LIN {X 0,Y 182.799,Z 411.389,A -85,B 0,C 180,E1 -25534.202,E2 -25534.202} C_VEL
LIN {X 0,Y 178.452,Z 402.819,A -85,B 0,C 180,E1 -25537.343,E2 -25537.343} C_VEL
LIN {X 0,Y 174.353,Z 395.574,A -85,B 0,C 180,E1 -25540.73,E2 -25540.73} C_VEL
LIN {X 0,Y 170.79,Z 389.828,A -85,B 0,C 180,E1 -25544.18,E2 -25544.18} C_VEL
LIN {X 0,Y 168.295,Z 385.886,A -85,B 0,C 180,E1 -25547.081,E2 -25547.081} C_VEL
LIN {X 0,Y 165.87,Z 382.031,A -85,B 0,C 180,E1 -25550.551,E2 -25550.551} C_VEL
LIN {X 0,Y 163.815,Z 378.873,A -85,B 0,C 180,E1 -25554.423,E2 -25554.423} C_VEL
LIN {X 0,Y 163.406,Z 377.726,A -85,B 0,C 180,E1 -25555.53,E2 -25555.53} C_VEL
LIN {X 0,Y 161.705,Z 376.148,A -85,B 0,C 180,E1 -25561.556,E2 -25561.556} C_VEL
LIN {X 0,Y 161.787,Z 376.62,A -85,B 0,C 180,E1 -25568.746,E2 -25568.746} C_VEL
LIN {X 0,Y 163.31,Z 378.032,A -85,B 0,C 180,E1 -25573.883,E2 -25573.883} C_VEL
LIN {X 0,Y 164.977,Z 381.356,A -85,B 0,C 180,E1 -25577.59,E2 -25577.59} C_VEL
LIN {X 0,Y 166.397,Z 382.961,A -85,B 0,C 180,E1 -25579.829,E2 -25579.829} C_VEL
LIN {X 0,Y 169.118,Z 387.647,A -85,B 0,C 180,E1 -25583.533,E2 -25583.533} C_VEL
LIN {X 0,Y 171.719,Z 392.777,A -85,B 0,C 180,E1 -25586.48,E2 -25586.48} C_VEL
LIN {X 0,Y 174.969,Z 399.659,A -85,B 0,C 180,E1 -25589.641,E2 -25589.641} C_VEL
LIN {X 0,Y 178.784,Z 408.58,A -85,B 0,C 180,E1 -25592.879,E2 -25592.879} C_VEL
LIN {X 0,Y 182.303,Z 418.101,A -85,B 0,C 180,E1 -25595.582,E2 -25595.582} C_VEL
LIN {X 0,Y 180.18,Z 440.666,A -85,B 0,C 180,E1 -25596.357,E2 -25596.357} C_VEL
LIN {X 0,Y 177.692,Z 453.902,A -85,B 0,C 180,E1 -25597.054,E2 -25597.054} C_VEL
LIN {X 0,Y 174.058,Z 466.777,A -85,B 0,C 180,E1 -25598.06,E2 -25598.06} C_VEL
LIN {X 0,Y 169.465,Z 479.095,A -85,B 0,C 180,E1 -25599.428,E2 -25599.428} C_VEL
LIN {X 0,Y 165.043,Z 488.832,A -85,B 0,C 180,E1 -25600.9,E2 -25600.9} C_VEL
LIN {X 0,Y 159.537,Z 499.053,A -85,B 0,C 180,E1 -25602.914,E2 -25602.914} C_VEL
LIN {X 0,Y 153.083,Z 509.068,A -85,B 0,C 180,E1 -25605.562,E2 -25605.562} C_VEL
LIN {X 0,Y 146.57,Z 517.891,A -85,B 0,C 180,E1 -25608.752,E2 -25608.752} C_VEL
LIN {X 0,Y 140.532,Z 524.996,A -85,B 0,C 180,E1 -25612.22,E2 -25612.22} C_VEL
LIN {X 0,Y 134.921,Z 530.971,A -85,B 0,C 180,E1 -25616.262,E2 -25616.262} C_VEL
LIN {X 0,Y 129.964,Z 535.823,A -85,B 0,C 180,E1 -25620.876,E2 -25620.876} C_VEL
LIN {X 0,Y 127.296,Z 538.125,A -85,B 0,C 180,E1 -25623.788,E2 -25623.788} C_VEL
LIN {X 0,Y 125.021,Z 540.003,A -85,B 0,C 180,E1 -25626.826,E2 -25626.826} C_VEL
LIN {X 0,Y 123.066,Z 541.427,A -85,B 0,C 180,E1 -25629.961,E2 -25629.961} C_VEL
LIN {X 0,Y 120.543,Z 543.117,A -85,B 0,C 180,E1 -25636.513,E2 -25636.513} C_VEL
LIN {X 0,Y 119.833,Z 543.394,A -85,B 0,C 180,E1 -25639.865,E2 -25639.865} C_VEL
LIN {X 0,Y 119.419,Z 543.249,A -85,B 0,C 180,E1 -25643.239,E2 -25643.239} C_VEL
LIN {X 0,Y 119.354,Z 542.709,A -85,B 0,C 180,E1 -25646.623,E2 -25646.623} C_VEL
LIN {X 0,Y 119.48,Z 541.653,A -85,B 0,C 180,E1 -25650.377,E2 -25650.377} C_VEL
LIN {X 0,Y 119.363,Z 540.421,A -85,B 0,C 180,E1 -25653.374,E2 -25653.374} C_VEL
LIN {X 0,Y 119.606,Z 537.522,A -85,B 0,C 180,E1 -25658.446,E2 -25658.446} C_VEL
LIN {X 0,Y 120.419,Z 533.561,A -85,B 0,C 180,E1 -25663.499,E2 -25663.499} C_VEL
LIN {X 0,Y 122.359,Z 527.446,A -85,B 0,C 180,E1 -25669.284,E2 -25669.284} C_VEL
LIN {X 0,Y 124.971,Z 520.737,A -85,B 0,C 180,E1 -25674.06,E2 -25674.06} C_VEL
LIN {X 0,Y 126.931,Z 516.144,A -85,B 0,C 180,E1 -25676.705,E2 -25676.705} C_VEL
LIN {X 0,Y 127.743,Z 512.422,A -85,B 0,C 180,E1 -25678.739,E2 -25678.739} C_VEL
LIN {X 0,Y 127.797,Z 505.991,A -85,B 0,C 180,E1 -25682.117,E2 -25682.117} C_VEL
LIN {X 0,Y 127.996,Z 499.009,A -85,B 0,C 180,E1 -25685.265,E2 -25685.265} C_VEL
LIN {X 0,Y 128.979,Z 494.425,A -85,B 0,C 180,E1 -25686.871,E2 -25686.871} C_VEL
LIN {X 0,Y 133.124,Z 482.951,A -85,B 0,C 180,E1 -25689.798,E2 -25689.798} C_VEL
LIN {X 0,Y 136.538,Z 471.516,A -85,B 0,C 180,E1 -25691.999,E2 -25691.999} C_VEL
LIN {X 0,Y 139.394,Z 459.785,A -85,B 0,C 180,E1 -25693.636,E2 -25693.636} C_VEL
LIN {X 0,Y 141.652,Z 446.808,A -85,B 0,C 180,E1 -25694.907,E2 -25694.907} C_VEL
LIN {X 0,Y 143.079,Z 433.332,A -85,B 0,C 180,E1 -25695.737,E2 -25695.737} C_VEL
LIN {X 0,Y 145.458,Z 398.287,A -85,B 0,C 180,E1 -25697.199,E2 -25697.199} C_VEL
LIN {X 0,Y 144.883,Z 389.327,A -85,B 0,C 180,E1 -25698.004,E2 -25698.004} C_VEL
LIN {X 0,Y 140.812,Z 377.368,A -85,B 0,C 180,E1 -25700.429,E2 -25700.429} C_VEL
LIN {X 0,Y 136.37,Z 367.095,A -85,B 0,C 180,E1 -25703.15,E2 -25703.15} C_VEL
LIN {X 0,Y 133.489,Z 362.113,A -85,B 0,C 180,E1 -25704.958,E2 -25704.958} C_VEL
LIN {X 0,Y 129.04,Z 355.347,A -85,B 0,C 180,E1 -25707.982,E2 -25707.982} C_VEL
LIN {X 0,Y 126.092,Z 351.147,A -85,B 0,C 180,E1 -25710.209,E2 -25710.209} C_VEL
LIN {X 0,Y 123.61,Z 347.782,A -85,B 0,C 180,E1 -25712.256,E2 -25712.256} C_VEL
LIN {X 0,Y 122.782,Z 346.727,A -85,B 0,C 180,E1 -25712.977,E2 -25712.977} C_VEL
LIN {X 0,Y 120.458,Z 344.175,A -85,B 0,C 180,E1 -25715.091,E2 -25715.091} C_VEL
LIN {X 0,Y 119.301,Z 341.838,A -85,B 0,C 180,E1 -25716.359,E2 -25716.359} C_VEL
LIN {X 0,Y 116.692,Z 339.986,A -85,B 0,C 180,E1 -25719.047,E2 -25719.047} C_VEL
LIN {X 0,Y 115.292,Z 337.525,A -85,B 0,C 180,E1 -25720.873,E2 -25720.873} C_VEL
LIN {X 0,Y 114.986,Z 336.158,A -85,B 0,C 180,E1 -25721.514,E2 -25721.514} C_VEL
LIN {X 0,Y 115.282,Z 336.094,A -85,B 0,C 180,E1 -25727.262,E2 -25727.262} C_VEL
LIN {X 0,Y 115.385,Z 336.109,A -85,B 0,C 180,E1 -25733.002,E2 -25733.002} C_VEL
LIN {X 0,Y 115.988,Z 336,A -85,B 0,C 180,E1 -25739.999,E2 -25739.999} C_VEL
LIN {X 0,Y 115.355,Z 336.095,A -85,B 0,C 180,E1 -25746.998,E2 -25746.998} C_VEL
LIN {X 0,Y 115.245,Z 336.108,A -85,B 0,C 180,E1 -25752.657,E2 -25752.657} C_VEL
LIN {X 0,Y 114.996,Z 336.138,A -85,B 0,C 180,E1 -25757.792,E2 -25757.792} C_VEL
LIN {X 0,Y 114.943,Z 336.152,A -85,B 0,C 180,E1 -25763.492,E2 -25763.492} C_VEL
LIN {X 0,Y 114.878,Z 336.207,A -85,B 0,C 180,E1 -25769.051,E2 -25769.051} C_VEL
LIN {X 0,Y 115.585,Z 338.454,A -85,B 0,C 180,E1 -25770.171,E2 -25770.171} C_VEL
LIN {X 0,Y 117.375,Z 340.759,A -85,B 0,C 180,E1 -25772.319,E2 -25772.319} C_VEL
LIN {X 0,Y 119.339,Z 342.102,A -85,B 0,C 180,E1 -25774.3,E2 -25774.3} C_VEL
LIN {X 0,Y 121.209,Z 345.34,A -85,B 0,C 180,E1 -25776.249,E2 -25776.249} C_VEL
LIN {X 0,Y 123.407,Z 347.522,A -85,B 0,C 180,E1 -25778.163,E2 -25778.163} C_VEL
LIN {X 0,Y 125.883,Z 351.047,A -85,B 0,C 180,E1 -25780.238,E2 -25780.238} C_VEL
LIN {X 0,Y 127.309,Z 353.048,A -85,B 0,C 180,E1 -25781.347,E2 -25781.347} C_VEL
LIN {X 0,Y 130.512,Z 357.56,A -85,B 0,C 180,E1 -25783.655,E2 -25783.655} C_VEL
LIN {X 0,Y 135.571,Z 365.369,A -85,B 0,C 180,E1 -25786.929,E2 -25786.929} C_VEL
LIN {X 0,Y 140.03,Z 373.18,A -85,B 0,C 180,E1 -25789.535,E2 -25789.535} C_VEL
LIN {X 0,Y 145.399,Z 384.296,A -85,B 0,C 180,E1 -25792.444,E2 -25792.444} C_VEL
LIN {X 0,Y 146.229,Z 386.228,A -85,B 0,C 180,E1 -25792.877,E2 -25792.877} C_VEL
LIN {X 0,Y 143.016,Z 431.95,A -85,B 0,C 180,E1 -25794.862,E2 -25794.862} C_VEL
LIN {X 0,Y 141.276,Z 445.448,A -85,B 0,C 180,E1 -25795.98,E2 -25795.98} C_VEL
LIN {X 0,Y 138.966,Z 457.681,A -85,B 0,C 180,E1 -25797.499,E2 -25797.499} C_VEL
LIN {X 0,Y 136.013,Z 468.763,A -85,B 0,C 180,E1 -25799.321,E2 -25799.321} C_VEL
LIN {X 0,Y 132.218,Z 480.314,A -85,B 0,C 180,E1 -25801.854,E2 -25801.854} C_VEL
LIN {X 0,Y 128.453,Z 490.68,A -85,B 0,C 180,E1 -25804.913,E2 -25804.913} C_VEL
LIN {X 0,Y 124.639,Z 500.01,A -85,B 0,C 180,E1 -25808.501,E2 -25808.501} C_VEL
LIN {X 0,Y 120.705,Z 509.025,A -85,B 0,C 180,E1 -25813.076,E2 -25813.076} C_VEL
LIN {X 0,Y 117.573,Z 516.285,A -85,B 0,C 180,E1 -25817.925,E2 -25817.925} C_VEL
LIN {X 0,Y 115.17,Z 522.106,A -85,B 0,C 180,E1 -25822.991,E2 -25822.991} C_VEL
LIN {X 0,Y 113.537,Z 526.693,A -85,B 0,C 180,E1 -25828.228,E2 -25828.228} C_VEL
LIN {X 0,Y 112.689,Z 530.291,A -85,B 0,C 180,E1 -25833.758,E2 -25833.758} C_VEL
LIN {X 0,Y 112.087,Z 533.325,A -85,B 0,C 180,E1 -25840.843,E2 -25840.843} C_VEL
LIN {X 0,Y 112.309,Z 534.286,A -85,B 0,C 180,E1 -25844.497,E2 -25844.497} C_VEL
LIN {X 0,Y 112.946,Z 534.841,A -85,B 0,C 180,E1 -25848.128,E2 -25848.128} C_VEL
LIN {X 0,Y 114.191,Z 534.925,A -85,B 0,C 180,E1 -25852.604,E2 -25852.604} C_VEL
LIN {X 0,Y 116.816,Z 534.015,A -85,B 0,C 180,E1 -25858.772,E2 -25858.772} C_VEL
LIN {X 0,Y 118.859,Z 532.918,A -85,B 0,C 180,E1 -25862.153,E2 -25862.153} C_VEL
LIN {X 0,Y 121.992,Z 530.899,A -85,B 0,C 180,E1 -25866.241,E2 -25866.241} C_VEL
LIN {X 0,Y 127.137,Z 526.951,A -85,B 0,C 180,E1 -25871.557,E2 -25871.557} C_VEL
LIN {X 0,Y 132.391,Z 522.293,A -85,B 0,C 180,E1 -25875.78,E2 -25875.78} C_VEL
LIN {X 0,Y 139.326,Z 515.206,A -85,B 0,C 180,E1 -25880.288,E2 -25880.288} C_VEL
LIN {X 0,Y 145.936,Z 507.482,A -85,B 0,C 180,E1 -25883.771,E2 -25883.771} C_VEL
LIN {X 0,Y 151.788,Z 499.51,A -85,B 0,C 180,E1 -25886.453,E2 -25886.453} C_VEL
LIN {X 0,Y 157.898,Z 489.721,A -85,B 0,C 180,E1 -25888.961,E2 -25888.961} C_VEL
LIN {X 0,Y 163.569,Z 478.78,A -85,B 0,C 180,E1 -25891.098,E2 -25891.098} C_VEL
LIN {X 0,Y 168.238,Z 467.913,A -85,B 0,C 180,E1 -25892.645,E2 -25892.645} C_VEL
LIN {X 0,Y 172.134,Z 456.207,A -85,B 0,C 180,E1 -25893.927,E2 -25893.927} C_VEL
LIN {X 0,Y 175.292,Z 443.368,A -85,B 0,C 180,E1 -25894.947,E2 -25894.947} C_VEL
LIN {X 0,Y 177.371,Z 430.99,A -85,B 0,C 180,E1 -25895.563,E2 -25895.563} C_VEL
LIN {X 0,Y 178.918,Z 414.661,A -85,B 0,C 180,E1 -25896.081,E2 -25896.081} C_VEL
LIN {X 0,Y 175.33,Z 407.397,A -85,B 0,C 180,E1 -25898.931,E2 -25898.931} C_VEL
LIN {X 0,Y 171.86,Z 400.977,A -85,B 0,C 180,E1 -25902.063,E2 -25902.063} C_VEL
LIN {X 0,Y 168.77,Z 395.843,A -85,B 0,C 180,E1 -25905.3,E2 -25905.3} C_VEL
LIN {X 0,Y 166.638,Z 392.303,A -85,B 0,C 180,E1 -25907.981,E2 -25907.981} C_VEL
LIN {X 0,Y 164.603,Z 388.858,A -85,B 0,C 180,E1 -25911.097,E2 -25911.097} C_VEL
LIN {X 0,Y 162.545,Z 385.367,A -85,B 0,C 180,E1 -25915.327,E2 -25915.327} C_VEL
LIN {X 0,Y 162.246,Z 384.661,A -85,B 0,C 180,E1 -25916.18,E2 -25916.18} C_VEL
LIN {X 0,Y 160.874,Z 383.217,A -85,B 0,C 180,E1 -25921.295,E2 -25921.295} C_VEL
LIN {X 0,Y 160.921,Z 383.691,A -85,B 0,C 180,E1 -25928.793,E2 -25928.793} C_VEL
LIN {X 0,Y 162.192,Z 384.921,A -85,B 0,C 180,E1 -25933.309,E2 -25933.309} C_VEL
LIN {X 0,Y 163.988,Z 388.453,A -85,B 0,C 180,E1 -25937.458,E2 -25937.458} C_VEL
LIN {X 0,Y 165.013,Z 389.709,A -85,B 0,C 180,E1 -25939.153,E2 -25939.153} C_VEL
LIN {X 0,Y 167.294,Z 393.779,A -85,B 0,C 180,E1 -25942.485,E2 -25942.485} C_VEL
LIN {X 0,Y 169.827,Z 399.15,A -85,B 0,C 180,E1 -25945.591,E2 -25945.591} C_VEL
LIN {X 0,Y 172.909,Z 406.19,A -85,B 0,C 180,E1 -25948.803,E2 -25948.803} C_VEL
LIN {X 0,Y 176.384,Z 414.842,A -85,B 0,C 180,E1 -25951.951,E2 -25951.951} C_VEL
LIN {X 0,Y 178.488,Z 420.805,A -85,B 0,C 180,E1 -25953.71,E2 -25953.71} C_VEL
LIN {X 0,Y 176.512,Z 440.736,A -85,B 0,C 180,E1 -25954.409,E2 -25954.409} C_VEL
LIN {X 0,Y 174.008,Z 453.597,A -85,B 0,C 180,E1 -25955.075,E2 -25955.075} C_VEL
LIN {X 0,Y 170.502,Z 465.847,A -85,B 0,C 180,E1 -25956.008,E2 -25956.008} C_VEL
LIN {X 0,Y 165.751,Z 478.298,A -85,B 0,C 180,E1 -25957.342,E2 -25957.342} C_VEL
LIN {X 0,Y 161.104,Z 488.137,A -85,B 0,C 180,E1 -25958.759,E2 -25958.759} C_VEL
LIN {X 0,Y 155.419,Z 498.431,A -85,B 0,C 180,E1 -25960.761,E2 -25960.761} C_VEL
LIN {X 0,Y 149.319,Z 507.707,A -85,B 0,C 180,E1 -25963.151,E2 -25963.151} C_VEL
LIN {X 0,Y 142.423,Z 516.71,A -85,B 0,C 180,E1 -25966.302,E2 -25966.302} C_VEL
LIN {X 0,Y 136.002,Z 523.988,A -85,B 0,C 180,E1 -25969.762,E2 -25969.762} C_VEL
LIN {X 0,Y 130.25,Z 529.843,A -85,B 0,C 180,E1 -25973.591,E2 -25973.591} C_VEL
LIN {X 0,Y 125.312,Z 534.478,A -85,B 0,C 180,E1 -25977.804,E2 -25977.804} C_VEL
LIN {X 0,Y 120.937,Z 538.031,A -85,B 0,C 180,E1 -25982.295,E2 -25982.295} C_VEL
LIN {X 0,Y 118.507,Z 539.861,A -85,B 0,C 180,E1 -25985.471,E2 -25985.471} C_VEL
LIN {X 0,Y 114.806,Z 542.26,A -85,B 0,C 180,E1 -25992.176,E2 -25992.176} C_VEL
LIN {X 0,Y 112.816,Z 543.129,A -85,B 0,C 180,E1 -25999.228,E2 -25999.228} C_VEL
LIN {X 0,Y 112.263,Z 542.379,A -85,B 0,C 180,E1 -26006.41,E2 -26006.41} C_VEL
LIN {X 0,Y 112.41,Z 541.423,A -85,B 0,C 180,E1 -26009.999,E2 -26009.999} C_VEL
LIN {X 0,Y 112.27,Z 540.031,A -85,B 0,C 180,E1 -26013.588,E2 -26013.588} C_VEL
LIN {X 0,Y 112.553,Z 537.082,A -85,B 0,C 180,E1 -26018.979,E2 -26018.979} C_VEL
LIN {X 0,Y 113.468,Z 533.061,A -85,B 0,C 180,E1 -26024.343,E2 -26024.343} C_VEL
LIN {X 0,Y 115.654,Z 526.854,A -85,B 0,C 180,E1 -26030.45,E2 -26030.45} C_VEL
LIN {X 0,Y 118.479,Z 520.07,A -85,B 0,C 180,E1 -26035.47,E2 -26035.47} C_VEL
LIN {X 0,Y 120.744,Z 514.832,A -85,B 0,C 180,E1 -26038.584,E2 -26038.584} C_VEL
LIN {X 0,Y 124.163,Z 506.59,A -85,B 0,C 180,E1 -26042.527,E2 -26042.527} C_VEL
LIN {X 0,Y 128.102,Z 496.752,A -85,B 0,C 180,E1 -26046.139,E2 -26046.139} C_VEL
LIN {X 0,Y 128.979,Z 494.425,A -85,B 0,C 180,E1 -26046.871,E2 -26046.871} C_VEL
LIN {X 0,Y 129.981,Z 489.751,A -85,B 0,C 180,E1 -26048.385,E2 -26048.385} C_VEL
LIN {X 0,Y 130.427,Z 478.545,A -85,B 0,C 180,E1 -26051.998,E2 -26051.998} C_VEL
LIN {X 0,Y 131.039,Z 471.722,A -85,B 0,C 180,E1 -26053.733,E2 -26053.733} C_VEL
LIN {X 0,Y 131.799,Z 468.136,A -85,B 0,C 180,E1 -26054.384,E2 -26054.384} C_VEL
LIN {X 0,Y 134.561,Z 456.507,A -85,B 0,C 180,E1 -26055.9,E2 -26055.9} C_VEL
LIN {X 0,Y 136.748,Z 443.617,A -85,B 0,C 180,E1 -26057.066,E2 -26057.066} C_VEL
LIN {X 0,Y 138.1,Z 429.088,A -85,B 0,C 180,E1 -26057.849,E2 -26057.849} C_VEL
LIN {X 0,Y 140.249,Z 399.102,A -85,B 0,C 180,E1 -26059.112,E2 -26059.112} C_VEL
LIN {X 0,Y 139.764,Z 391.546,A -85,B 0,C 180,E1 -26059.845,E2 -26059.845} C_VEL
LIN {X 0,Y 136.189,Z 380.798,A -85,B 0,C 180,E1 -26062.177,E2 -26062.177} C_VEL
LIN {X 0,Y 132.284,Z 371.453,A -85,B 0,C 180,E1 -26064.803,E2 -26064.803} C_VEL
LIN {X 0,Y 128.572,Z 364.909,A -85,B 0,C 180,E1 -26067.388,E2 -26067.388} C_VEL
LIN {X 0,Y 123.204,Z 356.965,A -85,B 0,C 180,E1 -26071.578,E2 -26071.578} C_VEL
LIN {X 0,Y 120.254,Z 352.917,A -85,B 0,C 180,E1 -26074.235,E2 -26074.235} C_VEL
LIN {X 0,Y 117.75,Z 349.777,A -85,B 0,C 180,E1 -26076.744,E2 -26076.744} C_VEL
LIN {X 0,Y 116.931,Z 348.248,A -85,B 0,C 180,E1 -26077.702,E2 -26077.702} C_VEL
LIN {X 0,Y 114.396,Z 345.983,A -85,B 0,C 180,E1 -26080.601,E2 -26080.601} C_VEL
LIN {X 0,Y 112.753,Z 342.88,A -85,B 0,C 180,E1 -26083.011,E2 -26083.011} C_VEL
LIN {X 0,Y 110.318,Z 341.255,A -85,B 0,C 180,E1 -26086.679,E2 -26086.679} C_VEL
LIN {X 0,Y 108.645,Z 338.426,A -85,B 0,C 180,E1 -26090.223,E2 -26090.223} C_VEL
LIN {X 0,Y 108.294,Z 336.972,A -85,B 0,C 180,E1 -26091.485,E2 -26091.485} C_VEL
LIN {X 0,Y 108.914,Z 336.88,A -85,B 0,C 180,E1 -26099.999,E2 -26099.999} C_VEL
LIN {X 0,Y 108.295,Z 336.968,A -85,B 0,C 180,E1 -26107.457,E2 -26107.457} C_VEL
LIN {X 0,Y 108.166,Z 336.991,A -85,B 0,C 180,E1 -26112.947,E2 -26112.947} C_VEL
LIN {X 0,Y 107.935,Z 337.086,A -85,B 0,C 180,E1 -26118.507,E2 -26118.507} C_VEL
LIN {X 0,Y 108.493,Z 339.139,A -85,B 0,C 180,E1 -26120.252,E2 -26120.252} C_VEL
LIN {X 0,Y 110.772,Z 341.962,A -85,B 0,C 180,E1 -26124.743,E2 -26124.743} C_VEL
LIN {X 0,Y 112.832,Z 343.115,A -85,B 0,C 180,E1 -26127.723,E2 -26127.723} C_VEL
LIN {X 0,Y 114.487,Z 346.252,A -85,B 0,C 180,E1 -26130.13,E2 -26130.13} C_VEL
LIN {X 0,Y 117.162,Z 348.772,A -85,B 0,C 180,E1 -26133.176,E2 -26133.176} C_VEL
LIN {X 0,Y 119.418,Z 352.183,A -85,B 0,C 180,E1 -26135.589,E2 -26135.589} C_VEL
LIN {X 0,Y 120.903,Z 353.816,A -85,B 0,C 180,E1 -26136.971,E2 -26136.971} C_VEL
LIN {X 0,Y 124.336,Z 358.803,A -85,B 0,C 180,E1 -26139.982,E2 -26139.982} C_VEL
LIN {X 0,Y 127.719,Z 363.738,A -85,B 0,C 180,E1 -26142.597,E2 -26142.597} C_VEL
LIN {X 0,Y 132.879,Z 372.086,A -85,B 0,C 180,E1 -26146.145,E2 -26146.145} C_VEL
LIN {X 0,Y 137.922,Z 381.827,A -85,B 0,C 180,E1 -26149.265,E2 -26149.265} C_VEL
LIN {X 0,Y 140.92,Z 388.415,A -85,B 0,C 180,E1 -26150.994,E2 -26150.994} C_VEL
LIN {X 0,Y 137.765,Z 431.864,A -85,B 0,C 180,E1 -26152.923,E2 -26152.923} C_VEL
LIN {X 0,Y 135.883,Z 445.712,A -85,B 0,C 180,E1 -26154.08,E2 -26154.08} C_VEL
LIN {X 0,Y 133.291,Z 458.5,A -85,B 0,C 180,E1 -26155.702,E2 -26155.702} C_VEL
LIN {X 0,Y 129.968,Z 470.244,A -85,B 0,C 180,E1 -26157.726,E2 -26157.726} C_VEL
LIN {X 0,Y 126.005,Z 481.573,A -85,B 0,C 180,E1 -26160.331,E2 -26160.331} C_VEL
LIN {X 0,Y 122.09,Z 491.743,A -85,B 0,C 180,E1 -26163.507,E2 -26163.507} C_VEL
LIN {X 0,Y 118.063,Z 500.901,A -85,B 0,C 180,E1 -26167.238,E2 -26167.238} C_VEL
LIN {X 0,Y 113.94,Z 509.809,A -85,B 0,C 180,E1 -26172.038,E2 -26172.038} C_VEL
LIN {X 0,Y 110.662,Z 516.974,A -85,B 0,C 180,E1 -26177.158,E2 -26177.158} C_VEL
LIN {X 0,Y 108.104,Z 522.698,A -85,B 0,C 180,E1 -26182.53,E2 -26182.53} C_VEL
LIN {X 0,Y 106.447,Z 527.205,A -85,B 0,C 180,E1 -26188.11,E2 -26188.11} C_VEL
LIN {X 0,Y 105.567,Z 530.644,A -85,B 0,C 180,E1 -26193.819,E2 -26193.819} C_VEL
LIN {X 0,Y 105.055,Z 532.379,A -85,B 0,C 180,E1 -26197.69,E2 -26197.69} C_VEL
LIN {X 0,Y 104.998,Z 533.704,A -85,B 0,C 180,E1 -26201.585,E2 -26201.585} C_VEL
LIN {X 0,Y 105.322,Z 534.634,A -85,B 0,C 180,E1 -26205.482,E2 -26205.482} C_VEL
LIN {X 0,Y 106.071,Z 535.129,A -85,B 0,C 180,E1 -26209.348,E2 -26209.348} C_VEL
LIN {X 0,Y 107.289,Z 535.201,A -85,B 0,C 180,E1 -26213.5,E2 -26213.5} C_VEL
LIN {X 0,Y 110.485,Z 534.205,A -85,B 0,C 180,E1 -26220.591,E2 -26220.591} C_VEL
LIN {X 0,Y 112.759,Z 533.046,A -85,B 0,C 180,E1 -26224.123,E2 -26224.123} C_VEL
LIN {X 0,Y 115.751,Z 531.262,A -85,B 0,C 180,E1 -26227.879,E2 -26227.879} C_VEL
LIN {X 0,Y 120.049,Z 528.247,A -85,B 0,C 180,E1 -26232.319,E2 -26232.319} C_VEL
LIN {X 0,Y 125.453,Z 523.919,A -85,B 0,C 180,E1 -26236.743,E2 -26236.743} C_VEL
LIN {X 0,Y 131.545,Z 518.352,A -85,B 0,C 180,E1 -26240.778,E2 -26240.778} C_VEL
LIN {X 0,Y 138.205,Z 511.354,A -85,B 0,C 180,E1 -26244.453,E2 -26244.453} C_VEL
LIN {X 0,Y 145.264,Z 502.723,A -85,B 0,C 180,E1 -26247.689,E2 -26247.689} C_VEL
LIN {X 0,Y 151.723,Z 493.408,A -85,B 0,C 180,E1 -26250.289,E2 -26250.289} C_VEL
LIN {X 0,Y 157.531,Z 483.314,A -85,B 0,C 180,E1 -26252.461,E2 -26252.461} C_VEL
LIN {X 0,Y 162.918,Z 472.021,A -85,B 0,C 180,E1 -26254.226,E2 -26254.226} C_VEL
LIN {X 0,Y 167.338,Z 460.287,A -85,B 0,C 180,E1 -26255.622,E2 -26255.622} C_VEL
LIN {X 0,Y 170.766,Z 448.312,A -85,B 0,C 180,E1 -26256.672,E2 -26256.672} C_VEL
LIN {X 0,Y 173.271,Z 435.759,A -85,B 0,C 180,E1 -26257.414,E2 -26257.414} C_VEL
LIN {X 0,Y 175.332,Z 418.304,A -85,B 0,C 180,E1 -26257.949,E2 -26257.949} C_VEL
LIN {X 0,Y 172.367,Z 411.99,A -85,B 0,C 180,E1 -26260.557,E2 -26260.557} C_VEL
LIN {X 0,Y 168.917,Z 405.563,A -85,B 0,C 180,E1 -26264,E2 -26264} C_VEL
LIN {X 0,Y 166.702,Z 401.685,A -85,B 0,C 180,E1 -26266.593,E2 -26266.593} C_VEL
LIN {X 0,Y 164.993,Z 398.634,A -85,B 0,C 180,E1 -26268.95,E2 -26268.95} C_VEL
LIN {X 0,Y 163.144,Z 395.409,A -85,B 0,C 180,E1 -26272.017,E2 -26272.017} C_VEL
LIN {X 0,Y 161.098,Z 391.549,A -85,B 0,C 180,E1 -26276.875,E2 -26276.875} C_VEL
LIN {X 0,Y 159.836,Z 390.177,A -85,B 0,C 180,E1 -26282.521,E2 -26282.521} C_VEL
LIN {X 0,Y 160.055,Z 390.765,A -85,B 0,C 180,E1 -26288.841,E2 -26288.841} C_VEL
LIN {X 0,Y 161.104,Z 391.812,A -85,B 0,C 180,E1 -26292.759,E2 -26292.759} C_VEL
LIN {X 0,Y 162.762,Z 395.265,A -85,B 0,C 180,E1 -26296.888,E2 -26296.888} C_VEL
LIN {X 0,Y 163.785,Z 396.679,A -85,B 0,C 180,E1 -26298.693,E2 -26298.693} C_VEL
LIN {X 0,Y 165.626,Z 400.165,A -85,B 0,C 180,E1 -26301.562,E2 -26301.562} C_VEL
LIN {X 0,Y 167.894,Z 405.33,A -85,B 0,C 180,E1 -26304.582,E2 -26304.582} C_VEL
LIN {X 0,Y 170.782,Z 412.392,A -85,B 0,C 180,E1 -26307.828,E2 -26307.828} C_VEL
LIN {X 0,Y 173.668,Z 420.159,A -85,B 0,C 180,E1 -26310.669,E2 -26310.669} C_VEL
LIN {X 0,Y 174.857,Z 423.716,A -85,B 0,C 180,E1 -26311.765,E2 -26311.765} C_VEL
LIN {X 0,Y 173.004,Z 441.112,A -85,B 0,C 180,E1 -26312.39,E2 -26312.39} C_VEL
LIN {X 0,Y 170.551,Z 453.173,A -85,B 0,C 180,E1 -26312.996,E2 -26312.996} C_VEL
LIN {X 0,Y 167.166,Z 464.912,A -85,B 0,C 180,E1 -26313.866,E2 -26313.866} C_VEL
LIN {X 0,Y 162.263,Z 477.507,A -85,B 0,C 180,E1 -26315.162,E2 -26315.162} C_VEL
LIN {X 0,Y 156.785,Z 488.729,A -85,B 0,C 180,E1 -26316.749,E2 -26316.749} C_VEL
LIN {X 0,Y 150.895,Z 498.851,A -85,B 0,C 180,E1 -26318.726,E2 -26318.726} C_VEL
LIN {X 0,Y 144.577,Z 507.983,A -85,B 0,C 180,E1 -26321.107,E2 -26321.107} C_VEL
LIN {X 0,Y 137.386,Z 516.896,A -85,B 0,C 180,E1 -26324.26,E2 -26324.26} C_VEL
LIN {X 0,Y 130.651,Z 524.094,A -85,B 0,C 180,E1 -26327.746,E2 -26327.746} C_VEL
LIN {X 0,Y 124.605,Z 529.866,A -85,B 0,C 180,E1 -26331.652,E2 -26331.652} C_VEL
LIN {X 0,Y 119.338,Z 534.437,A -85,B 0,C 180,E1 -26335.98,E2 -26335.98} C_VEL
LIN {X 0,Y 114.675,Z 537.937,A -85,B 0,C 180,E1 -26340.639,E2 -26340.639} C_VEL
LIN {X 0,Y 112.071,Z 539.713,A -85,B 0,C 180,E1 -26343.96,E2 -26343.96} C_VEL
LIN {X 0,Y 108.026,Z 542.059,A -85,B 0,C 180,E1 -26351.016,E2 -26351.016} C_VEL
LIN {X 0,Y 106.74,Z 542.663,A -85,B 0,C 180,E1 -26354.729,E2 -26354.729} C_VEL
LIN {X 0,Y 105.83,Z 542.852,A -85,B 0,C 180,E1 -26358.507,E2 -26358.507} C_VEL
LIN {X 0,Y 105.181,Z 542.05,A -85,B 0,C 180,E1 -26366.167,E2 -26366.167} C_VEL
LIN {X 0,Y 105.335,Z 541.069,A -85,B 0,C 180,E1 -26369.999,E2 -26369.999} C_VEL
LIN {X 0,Y 105.189,Z 539.627,A -85,B 0,C 180,E1 -26373.83,E2 -26373.83} C_VEL
LIN {X 0,Y 105.526,Z 536.63,A -85,B 0,C 180,E1 -26379.583,E2 -26379.583} C_VEL
LIN {X 0,Y 106.553,Z 532.548,A -85,B 0,C 180,E1 -26385.296,E2 -26385.296} C_VEL
LIN {X 0,Y 109.011,Z 526.263,A -85,B 0,C 180,E1 -26391.758,E2 -26391.758} C_VEL
LIN {X 0,Y 112.082,Z 519.405,A -85,B 0,C 180,E1 -26397.038,E2 -26397.038} C_VEL
LIN {X 0,Y 113.965,Z 515.38,A -85,B 0,C 180,E1 -26399.559,E2 -26399.559} C_VEL
LIN {X 0,Y 116.695,Z 509.196,A -85,B 0,C 180,E1 -26402.82,E2 -26402.82} C_VEL
LIN {X 0,Y 120.683,Z 500.042,A -85,B 0,C 180,E1 -26406.647,E2 -26406.647} C_VEL
LIN {X 0,Y 124.706,Z 489.923,A -85,B 0,C 180,E1 -26409.869,E2 -26409.869} C_VEL
LIN {X 0,Y 128.699,Z 478.671,A -85,B 0,C 180,E1 -26412.512,E2 -26412.512} C_VEL
LIN {X 0,Y 131.799,Z 468.136,A -85,B 0,C 180,E1 -26414.384,E2 -26414.384} C_VEL
LIN {X 0,Y 132.665,Z 462.724,A -85,B 0,C 180,E1 -26415.344,E2 -26415.344} C_VEL
LIN {X 0,Y 132.409,Z 453.764,A -85,B 0,C 180,E1 -26417.214,E2 -26417.214} C_VEL
LIN {X 0,Y 131.857,Z 444.61,A -85,B 0,C 180,E1 -26418.866,E2 -26418.866} C_VEL
LIN {X 0,Y 132.148,Z 438.863,A -85,B 0,C 180,E1 -26419.443,E2 -26419.443} C_VEL
LIN {X 0,Y 135.166,Z 400.629,A -85,B 0,C 180,E1 -26421.128,E2 -26421.128} C_VEL
LIN {X 0,Y 134.874,Z 393.98,A -85,B 0,C 180,E1 -26421.764,E2 -26421.764} C_VEL
LIN {X 0,Y 131.49,Z 383.608,A -85,B 0,C 180,E1 -26424.203,E2 -26424.203} C_VEL
LIN {X 0,Y 127.847,Z 374.792,A -85,B 0,C 180,E1 -26426.916,E2 -26426.916} C_VEL
LIN {X 0,Y 123.215,Z 366.999,A -85,B 0,C 180,E1 -26430.538,E2 -26430.538} C_VEL
LIN {X 0,Y 120.137,Z 362.449,A -85,B 0,C 180,E1 -26433.244,E2 -26433.244} C_VEL
LIN {X 0,Y 117.838,Z 359.099,A -85,B 0,C 180,E1 -26435.505,E2 -26435.505} C_VEL
LIN {X 0,Y 115.279,Z 355.624,A -85,B 0,C 180,E1 -26438.308,E2 -26438.308} C_VEL
LIN {X 0,Y 114.397,Z 354.432,A -85,B 0,C 180,E1 -26439.371,E2 -26439.371} C_VEL
LIN {X 0,Y 111.953,Z 351.561,A -85,B 0,C 180,E1 -26442.562,E2 -26442.562} C_VEL
LIN {X 0,Y 110.826,Z 349.535,A -85,B 0,C 180,E1 -26444.364,E2 -26444.364} C_VEL
LIN {X 0,Y 108.505,Z 347.495,A -85,B 0,C 180,E1 -26448.321,E2 -26448.321} C_VEL
LIN {X 0,Y 107.036,Z 344.518,A -85,B 0,C 180,E1 -26451.979,E2 -26451.979} C_VEL
LIN {X 0,Y 106.705,Z 343.89,A -85,B 0,C 180,E1 -26452.953,E2 -26452.953} C_VEL
LIN {X 0,Y 104.856,Z 342.696,A -85,B 0,C 180,E1 -26459.999,E2 -26459.999} C_VEL
LIN {X 0,Y 105.075,Z 343.36,A -85,B 0,C 180,E1 -26472.158,E2 -26472.158} C_VEL
LIN {X 0,Y 106.571,Z 344.146,A -85,B 0,C 180,E1 -26477.386,E2 -26477.386} C_VEL
LIN {X 0,Y 107.564,Z 346.607,A -85,B 0,C 180,E1 -26480.31,E2 -26480.31} C_VEL
LIN {X 0,Y 109.848,Z 349.097,A -85,B 0,C 180,E1 -26484.764,E2 -26484.764} C_VEL
LIN {X 0,Y 111.023,Z 349.852,A -85,B 0,C 180,E1 -26486.555,E2 -26486.555} C_VEL
LIN {X 0,Y 112.975,Z 353.182,A -85,B 0,C 180,E1 -26489.499,E2 -26489.499} C_VEL
LIN {X 0,Y 115.007,Z 355.245,A -85,B 0,C 180,E1 -26491.958,E2 -26491.958} C_VEL
LIN {X 0,Y 117.655,Z 359.003,A -85,B 0,C 180,E1 -26494.916,E2 -26494.916} C_VEL
LIN {X 0,Y 121.315,Z 364.264,A -85,B 0,C 180,E1 -26498.431,E2 -26498.431} C_VEL
LIN {X 0,Y 125.767,Z 371.178,A -85,B 0,C 180,E1 -26502.11,E2 -26502.11} C_VEL
LIN {X 0,Y 130.763,Z 380.001,A -85,B 0,C 180,E1 -26505.719,E2 -26505.719} C_VEL
LIN {X 0,Y 135.623,Z 390.455,A -85,B 0,C 180,E1 -26508.898,E2 -26508.898} C_VEL
LIN {X 0,Y 135.813,Z 391.21,A -85,B 0,C 180,E1 -26509.04,E2 -26509.04} C_VEL
LIN {X 0,Y 132.666,Z 431.76,A -85,B 0,C 180,E1 -26510.833,E2 -26510.833} C_VEL
LIN {X 0,Y 130.812,Z 445.029,A -85,B 0,C 180,E1 -26511.935,E2 -26511.935} C_VEL
LIN {X 0,Y 128.349,Z 457.153,A -85,B 0,C 180,E1 -26513.455,E2 -26513.455} C_VEL
LIN {X 0,Y 125.109,Z 468.525,A -85,B 0,C 180,E1 -26515.337,E2 -26515.337} C_VEL
LIN {X 0,Y 120.887,Z 480.231,A -85,B 0,C 180,E1 -26517.963,E2 -26517.963} C_VEL
LIN {X 0,Y 116.682,Z 490.7,A -85,B 0,C 180,E1 -26521.195,E2 -26521.195} C_VEL
LIN {X 0,Y 112.387,Z 500.146,A -85,B 0,C 180,E1 -26525.034,E2 -26525.034} C_VEL
LIN {X 0,Y 107.899,Z 509.233,A -85,B 0,C 180,E1 -26530.005,E2 -26530.005} C_VEL
LIN {X 0,Y 104.283,Z 516.55,A -85,B 0,C 180,E1 -26535.363,E2 -26535.363} C_VEL
LIN {X 0,Y 101.048,Z 523.272,A -85,B 0,C 180,E1 -26542.006,E2 -26542.006} C_VEL
LIN {X 0,Y 99.356,Z 527.706,A -85,B 0,C 180,E1 -26547.975,E2 -26547.975} C_VEL
LIN {X 0,Y 98.395,Z 531.084,A -85,B 0,C 180,E1 -26554.097,E2 -26554.097} C_VEL
LIN {X 0,Y 97.921,Z 532.787,A -85,B 0,C 180,E1 -26558.254,E2 -26558.254} C_VEL
LIN {X 0,Y 97.938,Z 534.081,A -85,B 0,C 180,E1 -26562.433,E2 -26562.433} C_VEL
LIN {X 0,Y 98.375,Z 534.97,A -85,B 0,C 180,E1 -26566.606,E2 -26566.606} C_VEL
LIN {X 0,Y 100.457,Z 535.474,A -85,B 0,C 180,E1 -26574.567,E2 -26574.567} C_VEL
LIN {X 0,Y 102.168,Z 535.132,A -85,B 0,C 180,E1 -26578.786,E2 -26578.786} C_VEL
LIN {X 0,Y 104.264,Z 534.381,A -85,B 0,C 180,E1 -26582.634,E2 -26582.634} C_VEL
LIN {X 0,Y 109.592,Z 531.637,A -85,B 0,C 180,E1 -26589.688,E2 -26589.688} C_VEL
LIN {X 0,Y 114.763,Z 528.279,A -85,B 0,C 180,E1 -26594.77,E2 -26594.77} C_VEL
LIN {X 0,Y 120.58,Z 523.88,A -85,B 0,C 180,E1 -26599.264,E2 -26599.264} C_VEL
LIN {X 0,Y 127.046,Z 518.235,A -85,B 0,C 180,E1 -26603.334,E2 -26603.334} C_VEL
LIN {X 0,Y 134.1,Z 511.116,A -85,B 0,C 180,E1 -26606.987,E2 -26606.987} C_VEL
LIN {X 0,Y 141.71,Z 502.1,A -85,B 0,C 180,E1 -26610.269,E2 -26610.269} C_VEL
LIN {X 0,Y 148.252,Z 492.93,A -85,B 0,C 180,E1 -26612.731,E2 -26612.731} C_VEL
LIN {X 0,Y 154.284,Z 482.601,A -85,B 0,C 180,E1 -26614.872,E2 -26614.872} C_VEL
LIN {X 0,Y 159.764,Z 471.385,A -85,B 0,C 180,E1 -26616.528,E2 -26616.528} C_VEL
LIN {X 0,Y 164.107,Z 460.043,A -85,B 0,C 180,E1 -26617.834,E2 -26617.834} C_VEL
LIN {X 0,Y 167.787,Z 447.319,A -85,B 0,C 180,E1 -26618.884,E2 -26618.884} C_VEL
LIN {X 0,Y 170.335,Z 434.321,A -85,B 0,C 180,E1 -26619.593,E2 -26619.593} C_VEL
LIN {X 0,Y 171.87,Z 421.656,A -85,B 0,C 180,E1 -26619.97,E2 -26619.97} C_VEL
LIN {X 0,Y 168.557,Z 414.703,A -85,B 0,C 180,E1 -26623.265,E2 -26623.265} C_VEL
LIN {X 0,Y 165.476,Z 408.852,A -85,B 0,C 180,E1 -26626.9,E2 -26626.9} C_VEL
LIN {X 0,Y 163.485,Z 405.173,A -85,B 0,C 180,E1 -26629.786,E2 -26629.786} C_VEL
LIN {X 0,Y 161.959,Z 402.243,A -85,B 0,C 180,E1 -26632.52,E2 -26632.52} C_VEL
LIN {X 0,Y 160.113,Z 398.537,A -85,B 0,C 180,E1 -26637.17,E2 -26637.17} C_VEL
LIN {X 0,Y 158.963,Z 397.225,A -85,B 0,C 180,E1 -26642.535,E2 -26642.535} C_VEL
LIN {X 0,Y 159.189,Z 397.837,A -85,B 0,C 180,E1 -26648.89,E2 -26648.89} C_VEL
LIN {X 0,Y 160.098,Z 398.901,A -85,B 0,C 180,E1 -26652.446,E2 -26652.446} C_VEL
LIN {X 0,Y 161.709,Z 402.244,A -85,B 0,C 180,E1 -26656.607,E2 -26656.607} C_VEL
LIN {X 0,Y 162.451,Z 403.433,A -85,B 0,C 180,E1 -26658.013,E2 -26658.013} C_VEL
LIN {X 0,Y 163.955,Z 406.431,A -85,B 0,C 180,E1 -26660.547,E2 -26660.547} C_VEL
LIN {X 0,Y 166.071,Z 411.647,A -85,B 0,C 180,E1 -26663.623,E2 -26663.623} C_VEL
LIN {X 0,Y 168.97,Z 419.289,A -85,B 0,C 180,E1 -26667.123,E2 -26667.123} C_VEL
LIN {X 0,Y 171.43,Z 426.611,A -85,B 0,C 180,E1 -26669.736,E2 -26669.736} C_VEL
LIN {X 0,Y 169.67,Z 441.805,A -85,B 0,C 180,E1 -26670.303,E2 -26670.303} C_VEL
LIN {X 0,Y 167,Z 454.164,A -85,B 0,C 180,E1 -26670.936,E2 -26670.936} C_VEL
LIN {X 0,Y 163.341,Z 465.974,A -85,B 0,C 180,E1 -26671.812,E2 -26671.812} C_VEL
LIN {X 0,Y 158.303,Z 478.292,A -85,B 0,C 180,E1 -26673.073,E2 -26673.073} C_VEL
LIN {X 0,Y 152.671,Z 489.312,A -85,B 0,C 180,E1 -26674.628,E2 -26674.628} C_VEL
LIN {X 0,Y 146.574,Z 499.236,A -85,B 0,C 180,E1 -26676.569,E2 -26676.569} C_VEL
LIN {X 0,Y 140.013,Z 508.26,A -85,B 0,C 180,E1 -26678.919,E2 -26678.919} C_VEL
LIN {X 0,Y 132.543,Z 517.082,A -85,B 0,C 180,E1 -26682.068,E2 -26682.068} C_VEL
LIN {X 0,Y 125.491,Z 524.186,A -85,B 0,C 180,E1 -26685.568,E2 -26685.568} C_VEL
LIN {X 0,Y 119.108,Z 529.875,A -85,B 0,C 180,E1 -26689.528,E2 -26689.528} C_VEL
LIN {X 0,Y 114.101,Z 533.902,A -85,B 0,C 180,E1 -26693.399,E2 -26693.399} C_VEL
LIN {X 0,Y 108.527,Z 537.834,A -85,B 0,C 180,E1 -26698.796,E2 -26698.796} C_VEL
LIN {X 0,Y 103.262,Z 540.905,A -85,B 0,C 180,E1 -26705.897,E2 -26705.897} C_VEL
LIN {X 0,Y 99.864,Z 542.427,A -85,B 0,C 180,E1 -26713.649,E2 -26713.649} C_VEL
LIN {X 0,Y 98.873,Z 542.574,A -85,B 0,C 180,E1 -26717.686,E2 -26717.686} C_VEL
LIN {X 0,Y 98.091,Z 541.721,A -85,B 0,C 180,E1 -26725.89,E2 -26725.89} C_VEL
LIN {X 0,Y 98.246,Z 540.713,A -85,B 0,C 180,E1 -26729.999,E2 -26729.999} C_VEL
LIN {X 0,Y 98.1,Z 539.218,A -85,B 0,C 180,E1 -26734.107,E2 -26734.107} C_VEL
LIN {X 0,Y 98.502,Z 536.164,A -85,B 0,C 180,E1 -26740.273,E2 -26740.273} C_VEL
LIN {X 0,Y 99.685,Z 532.021,A -85,B 0,C 180,E1 -26746.378,E2 -26746.378} C_VEL
LIN {X 0,Y 102.417,Z 525.67,A -85,B 0,C 180,E1 -26753.238,E2 -26753.238} C_VEL
LIN {X 0,Y 105.789,Z 518.741,A -85,B 0,C 180,E1 -26758.791,E2 -26758.791} C_VEL
LIN {X 0,Y 109.095,Z 511.739,A -85,B 0,C 180,E1 -26763.124,E2 -26763.124} C_VEL
LIN {X 0,Y 113.213,Z 503.076,A -85,B 0,C 180,E1 -26767.246,E2 -26767.246} C_VEL
LIN {X 0,Y 117.78,Z 492.468,A -85,B 0,C 180,E1 -26771.022,E2 -26771.022} C_VEL
LIN {X 0,Y 121.917,Z 481.984,A -85,B 0,C 180,E1 -26773.766,E2 -26773.766} C_VEL
LIN {X 0,Y 125.705,Z 470.436,A -85,B 0,C 180,E1 -26776.038,E2 -26776.038} C_VEL
LIN {X 0,Y 128.848,Z 458.466,A -85,B 0,C 180,E1 -26777.709,E2 -26777.709} C_VEL
LIN {X 0,Y 131.4,Z 444.815,A -85,B 0,C 180,E1 -26779.027,E2 -26779.027} C_VEL
LIN {X 0,Y 132.148,Z 438.863,A -85,B 0,C 180,E1 -26779.443,E2 -26779.443} C_VEL
LIN {X 0,Y 132.384,Z 433.087,A -85,B 0,C 180,E1 -26779.947,E2 -26779.947} C_VEL
LIN {X 0,Y 129.86,Z 414.309,A -85,B 0,C 180,E1 -26782.533,E2 -26782.533} C_VEL
LIN {X 0,Y 129.782,Z 408.483,A -85,B 0,C 180,E1 -26783.015,E2 -26783.015} C_VEL
LIN {X 0,Y 130.311,Z 399.937,A -85,B 0,C 180,E1 -26783.452,E2 -26783.452} C_VEL
LIN {X 0,Y 130.047,Z 396.241,A -85,B 0,C 180,E1 -26783.888,E2 -26783.888} C_VEL
LIN {X 0,Y 127.245,Z 387.363,A -85,B 0,C 180,E1 -26786.135,E2 -26786.135} C_VEL
LIN {X 0,Y 124.293,Z 379.725,A -85,B 0,C 180,E1 -26788.582,E2 -26788.582} C_VEL
LIN {X 0,Y 120.098,Z 372.428,A -85,B 0,C 180,E1 -26792.174,E2 -26792.174} C_VEL
LIN {X 0,Y 116.967,Z 367.58,A -85,B 0,C 180,E1 -26795.218,E2 -26795.218} C_VEL
LIN {X 0,Y 115.126,Z 364.871,A -85,B 0,C 180,E1 -26797.215,E2 -26797.215} C_VEL
LIN {X 0,Y 112.382,Z 360.856,A -85,B 0,C 180,E1 -26800.595,E2 -26800.595} C_VEL
LIN {X 0,Y 109.933,Z 357.66,A -85,B 0,C 180,E1 -26804.115,E2 -26804.115} C_VEL
LIN {X 0,Y 109.174,Z 356.238,A -85,B 0,C 180,E1 -26805.443,E2 -26805.443} C_VEL
LIN {X 0,Y 106.819,Z 353.793,A -85,B 0,C 180,E1 -26809.934,E2 -26809.934} C_VEL
LIN {X 0,Y 105.46,Z 350.798,A -85,B 0,C 180,E1 -26813.913,E2 -26813.913} C_VEL
LIN {X 0,Y 103.97,Z 349.812,A -85,B 0,C 180,E1 -26819.999,E2 -26819.999} C_VEL
LIN {X 0,Y 104.277,Z 350.452,A -85,B 0,C 180,E1 -26832.55,E2 -26832.55} C_VEL
LIN {X 0,Y 105.34,Z 351.152,A -85,B 0,C 180,E1 -26836.471,E2 -26836.471} C_VEL
LIN {X 0,Y 106.894,Z 354.352,A -85,B 0,C 180,E1 -26840.946,E2 -26840.946} C_VEL
LIN {X 0,Y 109.386,Z 356.711,A -85,B 0,C 180,E1 -26845.548,E2 -26845.548} C_VEL
LIN {X 0,Y 111.551,Z 360.16,A -85,B 0,C 180,E1 -26848.942,E2 -26848.942} C_VEL
LIN {X 0,Y 112.937,Z 361.692,A -85,B 0,C 180,E1 -26850.732,E2 -26850.732} C_VEL
LIN {X 0,Y 116.399,Z 366.803,A -85,B 0,C 180,E1 -26854.784,E2 -26854.784} C_VEL
LIN {X 0,Y 120.542,Z 373.126,A -85,B 0,C 180,E1 -26858.819,E2 -26858.819} C_VEL
LIN {X 0,Y 125.777,Z 382.392,A -85,B 0,C 180,E1 -26863.164,E2 -26863.164} C_VEL
LIN {X 0,Y 130.283,Z 391.971,A -85,B 0,C 180,E1 -26866.471,E2 -26866.471} C_VEL
LIN {X 0,Y 130.795,Z 393.231,A -85,B 0,C 180,E1 -26866.833,E2 -26866.833} C_VEL
LIN {X 0,Y 127.63,Z 432.614,A -85,B 0,C 180,E1 -26868.642,E2 -26868.642} C_VEL
LIN {X 0,Y 125.598,Z 446.198,A -85,B 0,C 180,E1 -26869.813,E2 -26869.813} C_VEL
LIN {X 0,Y 122.999,Z 457.985,A -85,B 0,C 180,E1 -26871.323,E2 -26871.323} C_VEL
LIN {X 0,Y 119.351,Z 469.981,A -85,B 0,C 180,E1 -26873.403,E2 -26873.403} C_VEL
LIN {X 0,Y 114.947,Z 481.46,A -85,B 0,C 180,E1 -26876.09,E2 -26876.09} C_VEL
LIN {X 0,Y 110.542,Z 491.761,A -85,B 0,C 180,E1 -26879.43,E2 -26879.43} C_VEL
LIN {X 0,Y 105.993,Z 501.026,A -85,B 0,C 180,E1 -26883.414,E2 -26883.414} C_VEL
LIN {X 0,Y 101.256,Z 510.004,A -85,B 0,C 180,E1 -26888.632,E2 -26888.632} C_VEL
LIN {X 0,Y 97.437,Z 517.231,A -85,B 0,C 180,E1 -26894.309,E2 -26894.309} C_VEL
LIN {X 0,Y 94.913,Z 522.118,A -85,B 0,C 180,E1 -26899.334,E2 -26899.334} C_VEL
LIN {X 0,Y 92.708,Z 526.876,A -85,B 0,C 180,E1 -26905.654,E2 -26905.654} C_VEL
LIN {X 0,Y 91.482,Z 530.876,A -85,B 0,C 180,E1 -26912.929,E2 -26912.929} C_VEL
LIN {X 0,Y 90.795,Z 533.193,A -85,B 0,C 180,E1 -26918.907,E2 -26918.907} C_VEL
LIN {X 0,Y 90.916,Z 534.456,A -85,B 0,C 180,E1 -26923.411,E2 -26923.411} C_VEL
LIN {X 0,Y 91.476,Z 535.287,A -85,B 0,C 180,E1 -26927.899,E2 -26927.899} C_VEL
LIN {X 0,Y 93.615,Z 535.751,A -85,B 0,C 180,E1 -26935.728,E2 -26935.728} C_VEL
LIN {X 0,Y 95.842,Z 535.357,A -85,B 0,C 180,E1 -26940.885,E2 -26940.885} C_VEL
LIN {X 0,Y 98.196,Z 534.544,A -85,B 0,C 180,E1 -26944.931,E2 -26944.931} C_VEL
LIN {X 0,Y 103.604,Z 531.993,A -85,B 0,C 180,E1 -26951.74,E2 -26951.74} C_VEL
LIN {X 0,Y 109.701,Z 528.312,A -85,B 0,C 180,E1 -26957.457,E2 -26957.457} C_VEL
LIN {X 0,Y 115.944,Z 523.841,A -85,B 0,C 180,E1 -26962.001,E2 -26962.001} C_VEL
LIN {X 0,Y 122.841,Z 518.114,A -85,B 0,C 180,E1 -26966.056,E2 -26966.056} C_VEL
LIN {X 0,Y 130.287,Z 510.867,A -85,B 0,C 180,E1 -26969.665,E2 -26969.665} C_VEL
LIN {X 0,Y 137.626,Z 502.523,A -85,B 0,C 180,E1 -26972.64,E2 -26972.64} C_VEL
LIN {X 0,Y 145.052,Z 492.424,A -85,B 0,C 180,E1 -26975.296,E2 -26975.296} C_VEL
LIN {X 0,Y 151.345,Z 481.88,A -85,B 0,C 180,E1 -26977.36,E2 -26977.36} C_VEL
LIN {X 0,Y 157.013,Z 470.442,A -85,B 0,C 180,E1 -26978.959,E2 -26978.959} C_VEL
LIN {X 0,Y 161.52,Z 458.739,A -85,B 0,C 180,E1 -26980.211,E2 -26980.211} C_VEL
LIN {X 0,Y 165.186,Z 445.763,A -85,B 0,C 180,E1 -26981.203,E2 -26981.203} C_VEL
LIN {X 0,Y 167.567,Z 433.42,A -85,B 0,C 180,E1 -26981.824,E2 -26981.824} C_VEL
LIN {X 0,Y 168.585,Z 425.309,A -85,B 0,C 180,E1 -26982.075,E2 -26982.075} C_VEL
LIN {X 0,Y 165.643,Z 418.845,A -85,B 0,C 180,E1 -26985.409,E2 -26985.409} C_VEL
LIN {X 0,Y 162.75,Z 413.089,A -85,B 0,C 180,E1 -26989.425,E2 -26989.425} C_VEL
LIN {X 0,Y 160.601,Z 408.849,A -85,B 0,C 180,E1 -26993.404,E2 -26993.404} C_VEL
LIN {X 0,Y 159.135,Z 405.501,A -85,B 0,C 180,E1 -26997.469,E2 -26997.469} C_VEL
LIN {X 0,Y 158.091,Z 404.273,A -85,B 0,C 180,E1 -27002.549,E2 -27002.549} C_VEL
LIN {X 0,Y 158.323,Z 404.917,A -85,B 0,C 180,E1 -27008.939,E2 -27008.939} C_VEL
LIN {X 0,Y 159.049,Z 405.835,A -85,B 0,C 180,E1 -27011.942,E2 -27011.942} C_VEL
LIN {X 0,Y 160.764,Z 409.389,A -85,B 0,C 180,E1 -27016.534,E2 -27016.534} C_VEL
LIN {X 0,Y 162.389,Z 412.807,A -85,B 0,C 180,E1 -27019.598,E2 -27019.598} C_VEL
LIN {X 0,Y 164.247,Z 417.793,A -85,B 0,C 180,E1 -27022.568,E2 -27022.568} C_VEL
LIN {X 0,Y 166.777,Z 425.097,A -85,B 0,C 180,E1 -27025.926,E2 -27025.926} C_VEL
LIN {X 0,Y 168.231,Z 429.704,A -85,B 0,C 180,E1 -27027.65,E2 -27027.65} C_VEL
LIN {X 0,Y 166.538,Z 442.647,A -85,B 0,C 180,E1 -27028.142,E2 -27028.142} C_VEL
LIN {X 0,Y 163.488,Z 455.626,A -85,B 0,C 180,E1 -27028.816,E2 -27028.816} C_VEL
LIN {X 0,Y 159.726,Z 467.03,A -85,B 0,C 180,E1 -27029.656,E2 -27029.656} C_VEL
LIN {X 0,Y 154.564,Z 479.078,A -85,B 0,C 180,E1 -27030.879,E2 -27030.879} C_VEL
LIN {X 0,Y 148.77,Z 489.839,A -85,B 0,C 180,E1 -27032.388,E2 -27032.388} C_VEL
LIN {X 0,Y 142.475,Z 499.62,A -85,B 0,C 180,E1 -27034.284,E2 -27034.284} C_VEL
LIN {X 0,Y 135.673,Z 508.537,A -85,B 0,C 180,E1 -27036.59,E2 -27036.59} C_VEL
LIN {X 0,Y 127.9,Z 517.266,A -85,B 0,C 180,E1 -27039.709,E2 -27039.709} C_VEL
LIN {X 0,Y 120.534,Z 524.259,A -85,B 0,C 180,E1 -27043.21,E2 -27043.21} C_VEL
LIN {X 0,Y 113.785,Z 529.879,A -85,B 0,C 180,E1 -27047.2,E2 -27047.2} C_VEL
LIN {X 0,Y 107.941,Z 534.215,A -85,B 0,C 180,E1 -27051.581,E2 -27051.581} C_VEL
LIN {X 0,Y 102.509,Z 537.719,A -85,B 0,C 180,E1 -27056.736,E2 -27056.736} C_VEL
LIN {X 0,Y 96.817,Z 540.733,A -85,B 0,C 180,E1 -27064.179,E2 -27064.179} C_VEL
LIN {X 0,Y 94.636,Z 541.66,A -85,B 0,C 180,E1 -27068.202,E2 -27068.202} C_VEL
LIN {X 0,Y 93.037,Z 542.178,A -85,B 0,C 180,E1 -27072.411,E2 -27072.411} C_VEL
LIN {X 0,Y 91.225,Z 542.032,A -85,B 0,C 180,E1 -27081.135,E2 -27081.135} C_VEL
LIN {X 0,Y 91.004,Z 541.389,A -85,B 0,C 180,E1 -27085.569,E2 -27085.569} C_VEL
LIN {X 0,Y 91.163,Z 540.343,A -85,B 0,C 180,E1 -27089.998,E2 -27089.998} C_VEL
LIN {X 0,Y 91.012,Z 538.805,A -85,B 0,C 180,E1 -27094.427,E2 -27094.427} C_VEL
LIN {X 0,Y 91.504,Z 535.693,A -85,B 0,C 180,E1 -27101.069,E2 -27101.069} C_VEL
LIN {X 0,Y 92.861,Z 531.487,A -85,B 0,C 180,E1 -27107.62,E2 -27107.62} C_VEL
LIN {X 0,Y 95.901,Z 525.068,A -85,B 0,C 180,E1 -27114.92,E2 -27114.92} C_VEL
LIN {X 0,Y 99.609,Z 518.059,A -85,B 0,C 180,E1 -27120.764,E2 -27120.764} C_VEL
LIN {X 0,Y 102.684,Z 511.861,A -85,B 0,C 180,E1 -27124.782,E2 -27124.782} C_VEL
LIN {X 0,Y 107.616,Z 502.161,A -85,B 0,C 180,E1 -27129.547,E2 -27129.547} C_VEL
LIN {X 0,Y 112.522,Z 491.421,A -85,B 0,C 180,E1 -27133.395,E2 -27133.395} C_VEL
LIN {X 0,Y 116.858,Z 480.76,A -85,B 0,C 180,E1 -27136.192,E2 -27136.192} C_VEL
LIN {X 0,Y 120.865,Z 468.857,A -85,B 0,C 180,E1 -27138.471,E2 -27138.471} C_VEL
LIN {X 0,Y 124.125,Z 456.44,A -85,B 0,C 180,E1 -27140.165,E2 -27140.165} C_VEL
LIN {X 0,Y 126.532,Z 443.691,A -85,B 0,C 180,E1 -27141.353,E2 -27141.353} C_VEL
LIN {X 0,Y 128.055,Z 429.422,A -85,B 0,C 180,E1 -27142.151,E2 -27142.151} C_VEL
LIN {X 0,Y 129.782,Z 408.483,A -85,B 0,C 180,E1 -27143.015,E2 -27143.015} C_VEL
LIN {X 0,Y 129.462,Z 404.774,A -85,B 0,C 180,E1 -27143.477,E2 -27143.477} C_VEL
LIN {X 0,Y 128.354,Z 401.484,A -85,B 0,C 180,E1 -27144.316,E2 -27144.316} C_VEL
LIN {X 0,Y 123.721,Z 392.62,A -85,B 0,C 180,E1 -27147.708,E2 -27147.708} C_VEL
LIN {X 0,Y 123.324,Z 391.509,A -85,B 0,C 180,E1 -27148.057,E2 -27148.057} C_VEL
LIN {X 0,Y 120.724,Z 384.377,A -85,B 0,C 180,E1 -27150.46,E2 -27150.46} C_VEL
LIN {X 0,Y 116.647,Z 377.13,A -85,B 0,C 180,E1 -27154.338,E2 -27154.338} C_VEL
LIN {X 0,Y 114.451,Z 373.514,A -85,B 0,C 180,E1 -27156.714,E2 -27156.714} C_VEL
LIN {X 0,Y 112.865,Z 371,A -85,B 0,C 180,E1 -27158.6,E2 -27158.6} C_VEL
LIN {X 0,Y 110.343,Z 367.173,A -85,B 0,C 180,E1 -27161.97,E2 -27161.97} C_VEL
LIN {X 0,Y 108.041,Z 363.857,A -85,B 0,C 180,E1 -27165.64,E2 -27165.64} C_VEL
LIN {X 0,Y 107.268,Z 362.691,A -85,B 0,C 180,E1 -27167.084,E2 -27167.084} C_VEL
LIN {X 0,Y 104.984,Z 359.559,A -85,B 0,C 180,E1 -27172.305,E2 -27172.305} C_VEL
LIN {X 0,Y 104.393,Z 357.818,A -85,B 0,C 180,E1 -27174.424,E2 -27174.424} C_VEL
LIN {X 0,Y 103.089,Z 356.9,A -85,B 0,C 180,E1 -27179.999,E2 -27179.999} C_VEL
LIN {X 0,Y 103.244,Z 357.414,A -85,B 0,C 180,E1 -27191.783,E2 -27191.783} C_VEL
LIN {X 0,Y 104.152,Z 358.037,A -85,B 0,C 180,E1 -27195.533,E2 -27195.533} C_VEL
LIN {X 0,Y 105.886,Z 361.523,A -85,B 0,C 180,E1 -27200.773,E2 -27200.773} C_VEL
LIN {X 0,Y 107.796,Z 363.497,A -85,B 0,C 180,E1 -27204.514,E2 -27204.514} C_VEL
LIN {X 0,Y 110.126,Z 367.091,A -85,B 0,C 180,E1 -27208.349,E2 -27208.349} C_VEL
LIN {X 0,Y 111.197,Z 368.601,A -85,B 0,C 180,E1 -27209.852,E2 -27209.852} C_VEL
LIN {X 0,Y 113.899,Z 372.704,A -85,B 0,C 180,E1 -27213.246,E2 -27213.246} C_VEL
LIN {X 0,Y 117.705,Z 378.896,A -85,B 0,C 180,E1 -27217.313,E2 -27217.313} C_VEL
LIN {X 0,Y 122.342,Z 387.47,A -85,B 0,C 180,E1 -27221.524,E2 -27221.524} C_VEL
LIN {X 0,Y 126.025,Z 395.711,A -85,B 0,C 180,E1 -27224.517,E2 -27224.517} C_VEL
LIN {X 0,Y 122.841,Z 433.186,A -85,B 0,C 180,E1 -27226.261,E2 -27226.261} C_VEL
LIN {X 0,Y 120.727,Z 446.551,A -85,B 0,C 180,E1 -27227.425,E2 -27227.425} C_VEL
LIN {X 0,Y 117.861,Z 458.784,A -85,B 0,C 180,E1 -27229.012,E2 -27229.012} C_VEL
LIN {X 0,Y 114.337,Z 469.843,A -85,B 0,C 180,E1 -27230.949,E2 -27230.949} C_VEL
LIN {X 0,Y 109.69,Z 481.398,A -85,B 0,C 180,E1 -27233.656,E2 -27233.656} C_VEL
LIN {X 0,Y 105.024,Z 491.753,A -85,B 0,C 180,E1 -27237.065,E2 -27237.065} C_VEL
LIN {X 0,Y 100.607,Z 500.241,A -85,B 0,C 180,E1 -27240.728,E2 -27240.728} C_VEL
LIN {X 0,Y 95.488,Z 509.418,A -85,B 0,C 180,E1 -27246.123,E2 -27246.123} C_VEL
LIN {X 0,Y 91.234,Z 516.798,A -85,B 0,C 180,E1 -27252.055,E2 -27252.055} C_VEL
LIN {X 0,Y 87.935,Z 522.722,A -85,B 0,C 180,E1 -27258.476,E2 -27258.476} C_VEL
LIN {X 0,Y 85.639,Z 527.406,A -85,B 0,C 180,E1 -27265.294,E2 -27265.294} C_VEL
LIN {X 0,Y 84.415,Z 531.041,A -85,B 0,C 180,E1 -27272.506,E2 -27272.506} C_VEL
LIN {X 0,Y 83.705,Z 533.598,A -85,B 0,C 180,E1 -27279.669,E2 -27279.669} C_VEL
LIN {X 0,Y 83.914,Z 534.825,A -85,B 0,C 180,E1 -27284.554,E2 -27284.554} C_VEL
LIN {X 0,Y 84.607,Z 535.603,A -85,B 0,C 180,E1 -27289.408,E2 -27289.408} C_VEL
LIN {X 0,Y 86.857,Z 536.025,A -85,B 0,C 180,E1 -27297.122,E2 -27297.122} C_VEL
LIN {X 0,Y 89.659,Z 535.568,A -85,B 0,C 180,E1 -27303.28,E2 -27303.28} C_VEL
LIN {X 0,Y 92.305,Z 534.707,A -85,B 0,C 180,E1 -27307.527,E2 -27307.527} C_VEL
LIN {X 0,Y 97.722,Z 532.365,A -85,B 0,C 180,E1 -27314.014,E2 -27314.014} C_VEL
LIN {X 0,Y 104.899,Z 528.345,A -85,B 0,C 180,E1 -27320.398,E2 -27320.398} C_VEL
LIN {X 0,Y 111.598,Z 523.799,A -85,B 0,C 180,E1 -27324.955,E2 -27324.955} C_VEL
LIN {X 0,Y 120.193,Z 516.835,A -85,B 0,C 180,E1 -27329.597,E2 -27329.597} C_VEL
LIN {X 0,Y 128.136,Z 509.246,A -85,B 0,C 180,E1 -27333.036,E2 -27333.036} C_VEL
LIN {X 0,Y 135.314,Z 501.123,A -85,B 0,C 180,E1 -27335.704,E2 -27335.704} C_VEL
LIN {X 0,Y 142.879,Z 490.784,A -85,B 0,C 180,E1 -27338.193,E2 -27338.193} C_VEL
LIN {X 0,Y 148.715,Z 481.164,A -85,B 0,C 180,E1 -27339.928,E2 -27339.928} C_VEL
LIN {X 0,Y 154.334,Z 469.976,A -85,B 0,C 180,E1 -27341.412,E2 -27341.412} C_VEL
LIN {X 0,Y 158.694,Z 458.858,A -85,B 0,C 180,E1 -27342.538,E2 -27342.538} C_VEL
LIN {X 0,Y 162.397,Z 446.101,A -85,B 0,C 180,E1 -27343.484,E2 -27343.484} C_VEL
LIN {X 0,Y 164.864,Z 433.696,A -85,B 0,C 180,E1 -27344.085,E2 -27344.085} C_VEL
LIN {X 0,Y 165.5,Z 429.031,A -85,B 0,C 180,E1 -27344.238,E2 -27344.238} C_VEL
LIN {X 0,Y 163.048,Z 423.471,A -85,B 0,C 180,E1 -27347.475,E2 -27347.475} C_VEL
LIN {X 0,Y 160.59,Z 418.199,A -85,B 0,C 180,E1 -27351.507,E2 -27351.507} C_VEL
LIN {X 0,Y 159.35,Z 415.564,A -85,B 0,C 180,E1 -27354.147,E2 -27354.147} C_VEL
LIN {X 0,Y 158.061,Z 412.417,A -85,B 0,C 180,E1 -27358.089,E2 -27358.089} C_VEL
LIN {X 0,Y 157.218,Z 411.321,A -85,B 0,C 180,E1 -27362.563,E2 -27362.563} C_VEL
LIN {X 0,Y 157.456,Z 411.998,A -85,B 0,C 180,E1 -27368.988,E2 -27368.988} C_VEL
LIN {X 0,Y 158.041,Z 412.842,A -85,B 0,C 180,E1 -27371.544,E2 -27371.544} C_VEL
LIN {X 0,Y 159.936,Z 417.019,A -85,B 0,C 180,E1 -27376.761,E2 -27376.761} C_VEL
LIN {X 0,Y 160.827,Z 419.116,A -85,B 0,C 180,E1 -27378.554,E2 -27378.554} C_VEL
LIN {X 0,Y 162.529,Z 424.1,A -85,B 0,C 180,E1 -27381.565,E2 -27381.565} C_VEL
LIN {X 0,Y 164.642,Z 430.883,A -85,B 0,C 180,E1 -27384.679,E2 -27384.679} C_VEL
LIN {X 0,Y 165.212,Z 432.877,A -85,B 0,C 180,E1 -27385.484,E2 -27385.484} C_VEL
LIN {X 0,Y 163.487,Z 444.038,A -85,B 0,C 180,E1 -27385.918,E2 -27385.918} C_VEL
LIN {X 0,Y 160.234,Z 456.989,A -85,B 0,C 180,E1 -27386.598,E2 -27386.598} C_VEL
LIN {X 0,Y 156.355,Z 468.083,A -85,B 0,C 180,E1 -27387.408,E2 -27387.408} C_VEL
LIN {X 0,Y 151.063,Z 479.803,A -85,B 0,C 180,E1 -27388.581,E2 -27388.581} C_VEL
LIN {X 0,Y 145.107,Z 490.354,A -85,B 0,C 180,E1 -27390.031,E2 -27390.031} C_VEL
LIN {X 0,Y 138.614,Z 500.004,A -85,B 0,C 180,E1 -27391.868,E2 -27391.868} C_VEL
LIN {X 0,Y 131.575,Z 508.813,A -85,B 0,C 180,E1 -27394.113,E2 -27394.113} C_VEL
LIN {X 0,Y 123.482,Z 517.429,A -85,B 0,C 180,E1 -27397.172,E2 -27397.172} C_VEL
LIN {X 0,Y 115.78,Z 524.33,A -85,B 0,C 180,E1 -27400.643,E2 -27400.643} C_VEL
LIN {X 0,Y 108.684,Z 529.882,A -85,B 0,C 180,E1 -27404.657,E2 -27404.657} C_VEL
LIN {X 0,Y 103.084,Z 533.76,A -85,B 0,C 180,E1 -27408.588,E2 -27408.588} C_VEL
LIN {X 0,Y 96.643,Z 537.603,A -85,B 0,C 180,E1 -27414.423,E2 -27414.423} C_VEL
LIN {X 0,Y 90.473,Z 540.562,A -85,B 0,C 180,E1 -27422.218,E2 -27422.218} C_VEL
LIN {X 0,Y 88.051,Z 541.453,A -85,B 0,C 180,E1 -27426.477,E2 -27426.477} C_VEL
LIN {X 0,Y 84.995,Z 542.015,A -85,B 0,C 180,E1 -27435.636,E2 -27435.636} C_VEL
LIN {X 0,Y 83.914,Z 541.057,A -85,B 0,C 180,E1 -27445.194,E2 -27445.194} C_VEL
LIN {X 0,Y 84.08,Z 539.959,A -85,B 0,C 180,E1 -27449.998,E2 -27449.998} C_VEL
LIN {X 0,Y 83.921,Z 538.391,A -85,B 0,C 180,E1 -27454.802,E2 -27454.802} C_VEL
LIN {X 0,Y 84.509,Z 535.219,A -85,B 0,C 180,E1 -27461.998,E2 -27461.998} C_VEL
LIN {X 0,Y 86.075,Z 530.95,A -85,B 0,C 180,E1 -27469.061,E2 -27469.061} C_VEL
LIN {X 0,Y 89.457,Z 524.463,A -85,B 0,C 180,E1 -27476.853,E2 -27476.853} C_VEL
LIN {X 0,Y 93.552,Z 517.351,A -85,B 0,C 180,E1 -27482.998,E2 -27482.998} C_VEL
LIN {X 0,Y 97.514,Z 510.068,A -85,B 0,C 180,E1 -27487.773,E2 -27487.773} C_VEL
LIN {X 0,Y 102.196,Z 501.237,A -85,B 0,C 180,E1 -27492.104,E2 -27492.104} C_VEL
LIN {X 0,Y 106.898,Z 491.553,A -85,B 0,C 180,E1 -27495.639,E2 -27495.639} C_VEL
LIN {X 0,Y 111.439,Z 480.974,A -85,B 0,C 180,E1 -27498.493,E2 -27498.493} C_VEL
LIN {X 0,Y 115.641,Z 469.261,A -85,B 0,C 180,E1 -27500.791,E2 -27500.791} C_VEL
LIN {X 0,Y 119.046,Z 457.05,A -85,B 0,C 180,E1 -27502.492,E2 -27502.492} C_VEL
LIN {X 0,Y 121.73,Z 443.72,A -85,B 0,C 180,E1 -27503.75,E2 -27503.75} C_VEL
LIN {X 0,Y 123.253,Z 430.601,A -85,B 0,C 180,E1 -27504.51,E2 -27504.51} C_VEL
LIN {X 0,Y 125.676,Z 401.5,A -85,B 0,C 180,E1 -27505.756,E2 -27505.756} C_VEL
LIN {X 0,Y 125.48,Z 398.664,A -85,B 0,C 180,E1 -27506.12,E2 -27506.12} C_VEL
LIN {X 0,Y 123.324,Z 391.509,A -85,B 0,C 180,E1 -27508.057,E2 -27508.057} C_VEL
LIN {X 0,Y 122.073,Z 388.605,A -85,B 0,C 180,E1 -27509.132,E2 -27509.132} C_VEL
LIN {X 0,Y 119.657,Z 385.228,A -85,B 0,C 180,E1 -27511.123,E2 -27511.123} C_VEL
LIN {X 0,Y 115.16,Z 381.324,A -85,B 0,C 180,E1 -27515.097,E2 -27515.097} C_VEL
LIN {X 0,Y 111.81,Z 378.5,A -85,B 0,C 180,E1 -27518.623,E2 -27518.623} C_VEL
LIN {X 0,Y 110.387,Z 376.778,A -85,B 0,C 180,E1 -27520.405,E2 -27520.405} C_VEL
LIN {X 0,Y 108.267,Z 373.364,A -85,B 0,C 180,E1 -27523.555,E2 -27523.555} C_VEL
LIN {X 0,Y 105.838,Z 369.434,A -85,B 0,C 180,E1 -27528.023,E2 -27528.023} C_VEL
LIN {X 0,Y 103.689,Z 366.22,A -85,B 0,C 180,E1 -27533.443,E2 -27533.443} C_VEL
LIN {X 0,Y 103.147,Z 364.685,A -85,B 0,C 180,E1 -27535.603,E2 -27535.603} C_VEL
LIN {X 0,Y 102.211,Z 363.981,A -85,B 0,C 180,E1 -27539.999,E2 -27539.999} C_VEL
LIN {X 0,Y 102.387,Z 364.472,A -85,B 0,C 180,E1 -27551.883,E2 -27551.883} C_VEL
LIN {X 0,Y 103.042,Z 365.118,A -85,B 0,C 180,E1 -27554.818,E2 -27554.818} C_VEL
LIN {X 0,Y 104.879,Z 368.691,A -85,B 0,C 180,E1 -27560.597,E2 -27560.597} C_VEL
LIN {X 0,Y 106.218,Z 370.203,A -85,B 0,C 180,E1 -27563.39,E2 -27563.39} C_VEL
LIN {X 0,Y 108.539,Z 373.808,A -85,B 0,C 180,E1 -27567.477,E2 -27567.477} C_VEL
LIN {X 0,Y 111.694,Z 378.98,A -85,B 0,C 180,E1 -27571.919,E2 -27571.919} C_VEL
LIN {X 0,Y 115.114,Z 384.925,A -85,B 0,C 180,E1 -27575.904,E2 -27575.904} C_VEL
LIN {X 0,Y 119.188,Z 392.957,A -85,B 0,C 180,E1 -27579.957,E2 -27579.957} C_VEL
LIN {X 0,Y 121.472,Z 398.319,A -85,B 0,C 180,E1 -27582.032,E2 -27582.032} C_VEL
LIN {X 0,Y 118.379,Z 433.099,A -85,B 0,C 180,E1 -27583.65,E2 -27583.65} C_VEL
LIN {X 0,Y 116.111,Z 446.744,A -85,B 0,C 180,E1 -27584.823,E2 -27584.823} C_VEL
LIN {X 0,Y 113.232,Z 458.508,A -85,B 0,C 180,E1 -27586.333,E2 -27586.333} C_VEL
LIN {X 0,Y 109.552,Z 469.705,A -85,B 0,C 180,E1 -27588.275,E2 -27588.275} C_VEL
LIN {X 0,Y 104.651,Z 481.336,A -85,B 0,C 180,E1 -27590.982,E2 -27590.982} C_VEL
LIN {X 0,Y 99.692,Z 491.748,A -85,B 0,C 180,E1 -27594.439,E2 -27594.439} C_VEL
LIN {X 0,Y 94.487,Z 501.145,A -85,B 0,C 180,E1 -27598.625,E2 -27598.625} C_VEL
LIN {X 0,Y 89.039,Z 510.19,A -85,B 0,C 180,E1 -27604.273,E2 -27604.273} C_VEL
LIN {X 0,Y 84.514,Z 517.48,A -85,B 0,C 180,E1 -27610.573,E2 -27610.573} C_VEL
LIN {X 0,Y 80.966,Z 523.327,A -85,B 0,C 180,E1 -27617.469,E2 -27617.469} C_VEL
LIN {X 0,Y 78.573,Z 527.935,A -85,B 0,C 180,E1 -27624.87,E2 -27624.87} C_VEL
LIN {X 0,Y 77.357,Z 531.229,A -85,B 0,C 180,E1 -27632.061,E2 -27632.061} C_VEL
LIN {X 0,Y 76.613,Z 534.004,A -85,B 0,C 180,E1 -27640.574,E2 -27640.574} C_VEL
LIN {X 0,Y 76.928,Z 535.177,A -85,B 0,C 180,E1 -27645.909,E2 -27645.909} C_VEL
LIN {X 0,Y 79.282,Z 536.269,A -85,B 0,C 180,E1 -27656.312,E2 -27656.312} C_VEL
LIN {X 0,Y 81.211,Z 536.234,A -85,B 0,C 180,E1 -27661.283,E2 -27661.283} C_VEL
LIN {X 0,Y 83.66,Z 535.764,A -85,B 0,C 180,E1 -27666.02,E2 -27666.02} C_VEL
LIN {X 0,Y 90.095,Z 533.573,A -85,B 0,C 180,E1 -27674.594,E2 -27674.594} C_VEL
LIN {X 0,Y 96.004,Z 530.787,A -85,B 0,C 180,E1 -27680.235,E2 -27680.235} C_VEL
LIN {X 0,Y 102.725,Z 526.936,A -85,B 0,C 180,E1 -27685.186,E2 -27685.186} C_VEL
LIN {X 0,Y 110.524,Z 521.617,A -85,B 0,C 180,E1 -27689.712,E2 -27689.712} C_VEL
LIN {X 0,Y 119.406,Z 514.294,A -85,B 0,C 180,E1 -27693.844,E2 -27693.844} C_VEL
LIN {X 0,Y 127.88,Z 505.99,A -85,B 0,C 180,E1 -27697.007,E2 -27697.007} C_VEL
LIN {X 0,Y 135.164,Z 497.438,A -85,B 0,C 180,E1 -27699.38,E2 -27699.38} C_VEL
LIN {X 0,Y 142.586,Z 486.778,A -85,B 0,C 180,E1 -27701.592,E2 -27701.592} C_VEL
LIN {X 0,Y 149.092,Z 475.421,A -85,B 0,C 180,E1 -27703.256,E2 -27703.256} C_VEL
LIN {X 0,Y 154.495,Z 463.302,A -85,B 0,C 180,E1 -27704.587,E2 -27704.587} C_VEL
LIN {X 0,Y 158.766,Z 450.615,A -85,B 0,C 180,E1 -27705.582,E2 -27705.582} C_VEL
LIN {X 0,Y 161.73,Z 438.122,A -85,B 0,C 180,E1 -27706.253,E2 -27706.253} C_VEL
LIN {X 0,Y 162.579,Z 432.907,A -85,B 0,C 180,E1 -27706.486,E2 -27706.486} C_VEL
LIN {X 0,Y 160.413,Z 427.528,A -85,B 0,C 180,E1 -27710.067,E2 -27710.067} C_VEL
LIN {X 0,Y 158.976,Z 424.245,A -85,B 0,C 180,E1 -27712.858,E2 -27712.858} C_VEL
LIN {X 0,Y 158.066,Z 422.146,A -85,B 0,C 180,E1 -27715.059,E2 -27715.059} C_VEL
LIN {X 0,Y 157.008,Z 419.316,A -85,B 0,C 180,E1 -27718.718,E2 -27718.718} C_VEL
LIN {X 0,Y 156.345,Z 418.372,A -85,B 0,C 180,E1 -27722.577,E2 -27722.577} C_VEL
LIN {X 0,Y 156.536,Z 418.99,A -85,B 0,C 180,E1 -27728.718,E2 -27728.718} C_VEL
LIN {X 0,Y 157.009,Z 419.764,A -85,B 0,C 180,E1 -27731.008,E2 -27731.008} C_VEL
LIN {X 0,Y 158.687,Z 423.755,A -85,B 0,C 180,E1 -27736.07,E2 -27736.07} C_VEL
LIN {X 0,Y 159.539,Z 426.099,A -85,B 0,C 180,E1 -27737.961,E2 -27737.961} C_VEL
LIN {X 0,Y 160.912,Z 430.53,A -85,B 0,C 180,E1 -27740.619,E2 -27740.619} C_VEL
LIN {X 0,Y 162.384,Z 436.278,A -85,B 0,C 180,E1 -27743.274,E2 -27743.274} C_VEL
LIN {X 0,Y 159.846,Z 449.089,A -85,B 0,C 180,E1 -27743.786,E2 -27743.786} C_VEL
LIN {X 0,Y 155.888,Z 462.241,A -85,B 0,C 180,E1 -27744.555,E2 -27744.555} C_VEL
LIN {X 0,Y 150.901,Z 474.346,A -85,B 0,C 180,E1 -27745.528,E2 -27745.528} C_VEL
LIN {X 0,Y 144.703,Z 485.959,A -85,B 0,C 180,E1 -27746.817,E2 -27746.817} C_VEL
LIN {X 0,Y 137.963,Z 496.399,A -85,B 0,C 180,E1 -27748.508,E2 -27748.508} C_VEL
LIN {X 0,Y 130.565,Z 505.836,A -85,B 0,C 180,E1 -27750.543,E2 -27750.543} C_VEL
LIN {X 0,Y 122.073,Z 514.934,A -85,B 0,C 180,E1 -27753.404,E2 -27753.404} C_VEL
LIN {X 0,Y 113.931,Z 522.286,A -85,B 0,C 180,E1 -27756.684,E2 -27756.684} C_VEL
LIN {X 0,Y 106.217,Z 528.207,A -85,B 0,C 180,E1 -27760.454,E2 -27760.454} C_VEL
LIN {X 0,Y 99.166,Z 532.901,A -85,B 0,C 180,E1 -27764.868,E2 -27764.868} C_VEL
LIN {X 0,Y 92.915,Z 536.51,A -85,B 0,C 180,E1 -27769.988,E2 -27769.988} C_VEL
LIN {X 0,Y 87.351,Z 539.134,A -85,B 0,C 180,E1 -27775.721,E2 -27775.721} C_VEL
LIN {X 0,Y 84.227,Z 540.39,A -85,B 0,C 180,E1 -27779.956,E2 -27779.956} C_VEL
LIN {X 0,Y 81.561,Z 541.233,A -85,B 0,C 180,E1 -27784.477,E2 -27784.477} C_VEL
LIN {X 0,Y 78.123,Z 541.736,A -85,B 0,C 180,E1 -27794.341,E2 -27794.341} C_VEL
LIN {X 0,Y 76.849,Z 540.718,A -85,B 0,C 180,E1 -27804.751,E2 -27804.751} C_VEL
LIN {X 0,Y 76.985,Z 539.574,A -85,B 0,C 180,E1 -27809.998,E2 -27809.998} C_VEL
LIN {X 0,Y 76.954,Z 537.029,A -85,B 0,C 180,E1 -27817.872,E2 -27817.872} C_VEL
LIN {X 0,Y 78.007,Z 533.443,A -85,B 0,C 180,E1 -27825.679,E2 -27825.679} C_VEL
LIN {X 0,Y 80.222,Z 528.718,A -85,B 0,C 180,E1 -27833.216,E2 -27833.216} C_VEL
LIN {X 0,Y 83.84,Z 522.736,A -85,B 0,C 180,E1 -27840.193,E2 -27840.193} C_VEL
LIN {X 0,Y 88.198,Z 515.549,A -85,B 0,C 180,E1 -27846.385,E2 -27846.385} C_VEL
LIN {X 0,Y 92.917,Z 507.603,A -85,B 0,C 180,E1 -27851.435,E2 -27851.435} C_VEL
LIN {X 0,Y 98.12,Z 498.344,A -85,B 0,C 180,E1 -27855.744,E2 -27855.744} C_VEL
LIN {X 0,Y 102.628,Z 489.31,A -85,B 0,C 180,E1 -27858.873,E2 -27858.873} C_VEL
LIN {X 0,Y 107.449,Z 478.159,A -85,B 0,C 180,E1 -27861.708,E2 -27861.708} C_VEL
LIN {X 0,Y 111.942,Z 465.667,A -85,B 0,C 180,E1 -27863.93,E2 -27863.93} C_VEL
LIN {X 0,Y 115.328,Z 453.015,A -85,B 0,C 180,E1 -27865.53,E2 -27865.53} C_VEL
LIN {X 0,Y 117.785,Z 439.399,A -85,B 0,C 180,E1 -27866.65,E2 -27866.65} C_VEL
LIN {X 0,Y 120.401,Z 412.541,A -85,B 0,C 180,E1 -27867.85,E2 -27867.85} C_VEL
LIN {X 0,Y 121.233,Z 401.625,A -85,B 0,C 180,E1 -27868.389,E2 -27868.389} C_VEL
LIN {X 0,Y 118.315,Z 391.786,A -85,B 0,C 180,E1 -27871.384,E2 -27871.384} C_VEL
LIN {X 0,Y 116.987,Z 388.579,A -85,B 0,C 180,E1 -27872.736,E2 -27872.736} C_VEL
LIN {X 0,Y 113.492,Z 381.935,A -85,B 0,C 180,E1 -27876.506,E2 -27876.506} C_VEL
LIN {X 0,Y 110.663,Z 377.164,A -85,B 0,C 180,E1 -27880.04,E2 -27880.04} C_VEL
LIN {X 0,Y 110.387,Z 376.778,A -85,B 0,C 180,E1 -27880.405,E2 -27880.405} C_VEL
LIN {X 0,Y 108.458,Z 374.562,A -85,B 0,C 180,E1 -27883.094,E2 -27883.094} C_VEL
LIN {X 0,Y 106.575,Z 373.212,A -85,B 0,C 180,E1 -27886.007,E2 -27886.007} C_VEL
LIN {X 0,Y 103.4,Z 372.07,A -85,B 0,C 180,E1 -27892.302,E2 -27892.302} C_VEL
LIN {X 0,Y 101.965,Z 371.59,A -85,B 0,C 180,E1 -27896.718,E2 -27896.718} C_VEL
LIN {X 0,Y 101.335,Z 371.041,A -85,B 0,C 180,E1 -27899.999,E2 -27899.999} C_VEL
LIN {X 0,Y 101.528,Z 371.552,A -85,B 0,C 180,E1 -27911.985,E2 -27911.985} C_VEL
LIN {X 0,Y 101.957,Z 372.125,A -85,B 0,C 180,E1 -27914.087,E2 -27914.087} C_VEL
LIN {X 0,Y 103.753,Z 375.684,A -85,B 0,C 180,E1 -27920.119,E2 -27920.119} C_VEL
LIN {X 0,Y 104.706,Z 376.949,A -85,B 0,C 180,E1 -27922.285,E2 -27922.285} C_VEL
LIN {X 0,Y 107.298,Z 381.309,A -85,B 0,C 180,E1 -27927.158,E2 -27927.158} C_VEL
LIN {X 0,Y 110.005,Z 386.017,A -85,B 0,C 180,E1 -27931.161,E2 -27931.161} C_VEL
LIN {X 0,Y 113.503,Z 392.76,A -85,B 0,C 180,E1 -27935.478,E2 -27935.478} C_VEL
LIN {X 0,Y 116.807,Z 400.123,A -85,B 0,C 180,E1 -27939.007,E2 -27939.007} C_VEL
LIN {X 0,Y 117.124,Z 400.959,A -85,B 0,C 180,E1 -27939.332,E2 -27939.332} C_VEL
LIN {X 0,Y 114.049,Z 433.846,A -85,B 0,C 180,E1 -27940.889,E2 -27940.889} C_VEL
LIN {X 0,Y 111.746,Z 447.001,A -85,B 0,C 180,E1 -27942.022,E2 -27942.022} C_VEL
LIN {X 0,Y 108.549,Z 459.309,A -85,B 0,C 180,E1 -27943.589,E2 -27943.589} C_VEL
LIN {X 0,Y 104.346,Z 471.16,A -85,B 0,C 180,E1 -27945.673,E2 -27945.673} C_VEL
LIN {X 0,Y 99.253,Z 482.565,A -85,B 0,C 180,E1 -27948.41,E2 -27948.41} C_VEL
LIN {X 0,Y 94.011,Z 492.806,A -85,B 0,C 180,E1 -27951.924,E2 -27951.924} C_VEL
LIN {X 0,Y 88.512,Z 502.019,A -85,B 0,C 180,E1 -27956.236,E2 -27956.236} C_VEL
LIN {X 0,Y 82.705,Z 510.961,A -85,B 0,C 180,E1 -27962.138,E2 -27962.138} C_VEL
LIN {X 0,Y 77.861,Z 518.161,A -85,B 0,C 180,E1 -27968.837,E2 -27968.837} C_VEL
LIN {X 0,Y 74.03,Z 523.918,A -85,B 0,C 180,E1 -27976.273,E2 -27976.273} C_VEL
LIN {X 0,Y 71.511,Z 528.447,A -85,B 0,C 180,E1 -27984.362,E2 -27984.362} C_VEL
LIN {X 0,Y 70.301,Z 531.382,A -85,B 0,C 180,E1 -27991.432,E2 -27991.432} C_VEL
LIN {X 0,Y 69.527,Z 534.408,A -85,B 0,C 180,E1 -28001.666,E2 -28001.666} C_VEL
LIN {X 0,Y 69.993,Z 535.522,A -85,B 0,C 180,E1 -28007.533,E2 -28007.533} C_VEL
LIN {X 0,Y 71.124,Z 536.233,A -85,B 0,C 180,E1 -28013.284,E2 -28013.284} C_VEL
LIN {X 0,Y 73.486,Z 536.576,A -85,B 0,C 180,E1 -28020.603,E2 -28020.603} C_VEL
LIN {X 0,Y 77.878,Z 535.958,A -85,B 0,C 180,E1 -28029.178,E2 -28029.178} C_VEL
LIN {X 0,Y 85.06,Z 533.705,A -85,B 0,C 180,E1 -28038.043,E2 -28038.043} C_VEL
LIN {X 0,Y 91.503,Z 530.854,A -85,B 0,C 180,E1 -28043.754,E2 -28043.754} C_VEL
LIN {X 0,Y 98.748,Z 526.933,A -85,B 0,C 180,E1 -28048.657,E2 -28048.657} C_VEL
LIN {X 0,Y 107.864,Z 520.897,A -85,B 0,C 180,E1 -28053.484,E2 -28053.484} C_VEL
LIN {X 0,Y 116.394,Z 514.093,A -85,B 0,C 180,E1 -28057.047,E2 -28057.047} C_VEL
LIN {X 0,Y 124.724,Z 506.188,A -85,B 0,C 180,E1 -28059.918,E2 -28059.918} C_VEL
LIN {X 0,Y 132.772,Z 496.968,A -85,B 0,C 180,E1 -28062.326,E2 -28062.326} C_VEL
LIN {X 0,Y 140.458,Z 486.151,A -85,B 0,C 180,E1 -28064.409,E2 -28064.409} C_VEL
LIN {X 0,Y 146.813,Z 475.253,A -85,B 0,C 180,E1 -28065.881,E2 -28065.881} C_VEL
LIN {X 0,Y 151.982,Z 463.964,A -85,B 0,C 180,E1 -28067.055,E2 -28067.055} C_VEL
LIN {X 0,Y 156.475,Z 451.064,A -85,B 0,C 180,E1 -28068.011,E2 -28068.011} C_VEL
LIN {X 0,Y 159.54,Z 438.568,A -85,B 0,C 180,E1 -28068.647,E2 -28068.647} C_VEL
LIN {X 0,Y 159.772,Z 436.999,A -85,B 0,C 180,E1 -28068.767,E2 -28068.767} C_VEL
LIN {X 0,Y 158.044,Z 431.833,A -85,B 0,C 180,E1 -28072.655,E2 -28072.655} C_VEL
LIN {X 0,Y 156.867,Z 428.815,A -85,B 0,C 180,E1 -28075.826,E2 -28075.826} C_VEL
LIN {X 0,Y 155.974,Z 426.21,A -85,B 0,C 180,E1 -28079.355,E2 -28079.355} C_VEL
LIN {X 0,Y 155.472,Z 425.423,A -85,B 0,C 180,E1 -28082.591,E2 -28082.591} C_VEL
LIN {X 0,Y 155.627,Z 426.005,A -85,B 0,C 180,E1 -28088.498,E2 -28088.498} C_VEL
LIN {X 0,Y 156.01,Z 426.721,A -85,B 0,C 180,E1 -28090.546,E2 -28090.546} C_VEL
LIN {X 0,Y 157.459,Z 430.467,A -85,B 0,C 180,E1 -28095.368,E2 -28095.368} C_VEL
LIN {X 0,Y 158.273,Z 433.333,A -85,B 0,C 180,E1 -28097.525,E2 -28097.525} C_VEL
LIN {X 0,Y 159.389,Z 438.302,A -85,B 0,C 180,E1 -28100.319,E2 -28100.319} C_VEL
LIN {X 0,Y 159.64,Z 439.734,A -85,B 0,C 180,E1 -28100.988,E2 -28100.988} C_VEL
LIN {X 0,Y 156.719,Z 452.434,A -85,B 0,C 180,E1 -28101.502,E2 -28101.502} C_VEL
LIN {X 0,Y 152.561,Z 464.795,A -85,B 0,C 180,E1 -28102.246,E2 -28102.246} C_VEL
LIN {X 0,Y 147.199,Z 476.713,A -85,B 0,C 180,E1 -28103.205,E2 -28103.205} C_VEL
LIN {X 0,Y 140.886,Z 487.838,A -85,B 0,C 180,E1 -28104.439,E2 -28104.439} C_VEL
LIN {X 0,Y 134.731,Z 496.846,A -85,B 0,C 180,E1 -28105.865,E2 -28105.865} C_VEL
LIN {X 0,Y 127.109,Z 506.121,A -85,B 0,C 180,E1 -28107.789,E2 -28107.789} C_VEL
LIN {X 0,Y 118.32,Z 515.12,A -85,B 0,C 180,E1 -28110.539,E2 -28110.539} C_VEL
LIN {X 0,Y 109.828,Z 522.394,A -85,B 0,C 180,E1 -28113.706,E2 -28113.706} C_VEL
LIN {X 0,Y 101.756,Z 528.243,A -85,B 0,C 180,E1 -28117.412,E2 -28117.412} C_VEL
LIN {X 0,Y 94.283,Z 532.873,A -85,B 0,C 180,E1 -28121.803,E2 -28121.803} C_VEL
LIN {X 0,Y 87.574,Z 536.423,A -85,B 0,C 180,E1 -28126.987,E2 -28126.987} C_VEL
LIN {X 0,Y 81.556,Z 538.99,A -85,B 0,C 180,E1 -28132.898,E2 -28132.898} C_VEL
LIN {X 0,Y 78.137,Z 540.214,A -85,B 0,C 180,E1 -28137.337,E2 -28137.337} C_VEL
LIN {X 0,Y 75.188,Z 541.007,A -85,B 0,C 180,E1 -28142.135,E2 -28142.135} C_VEL
LIN {X 0,Y 71.278,Z 541.457,A -85,B 0,C 180,E1 -28152.793,E2 -28152.793} C_VEL
LIN {X 0,Y 70.209,Z 541.116,A -85,B 0,C 180,E1 -28158.449,E2 -28158.449} C_VEL
LIN {X 0,Y 69.774,Z 540.363,A -85,B 0,C 180,E1 -28164.217,E2 -28164.217} C_VEL
LIN {X 0,Y 69.883,Z 539.188,A -85,B 0,C 180,E1 -28169.998,E2 -28169.998} C_VEL
LIN {X 0,Y 69.918,Z 536.586,A -85,B 0,C 180,E1 -28178.67,E2 -28178.67} C_VEL
LIN {X 0,Y 71.163,Z 532.939,A -85,B 0,C 180,E1 -28187.232,E2 -28187.232} C_VEL
LIN {X 0,Y 73.718,Z 528.149,A -85,B 0,C 180,E1 -28195.402,E2 -28195.402} C_VEL
LIN {X 0,Y 77.718,Z 522.092,A -85,B 0,C 180,E1 -28202.857,E2 -28202.857} C_VEL
LIN {X 0,Y 81.702,Z 516.162,A -85,B 0,C 180,E1 -28208.281,E2 -28208.281} C_VEL
LIN {X 0,Y 85.624,Z 510.075,A -85,B 0,C 180,E1 -28212.619,E2 -28212.619} C_VEL
LIN {X 0,Y 90.947,Z 501.367,A -85,B 0,C 180,E1 -28217.23,E2 -28217.23} C_VEL
LIN {X 0,Y 96.824,Z 490.63,A -85,B 0,C 180,E1 -28221.284,E2 -28221.284} C_VEL
LIN {X 0,Y 101.886,Z 479.967,A -85,B 0,C 180,E1 -28224.142,E2 -28224.142} C_VEL
LIN {X 0,Y 106.532,Z 468.071,A -85,B 0,C 180,E1 -28226.393,E2 -28226.393} C_VEL
LIN {X 0,Y 110.329,Z 455.376,A -85,B 0,C 180,E1 -28228.084,E2 -28228.084} C_VEL
LIN {X 0,Y 113.038,Z 442.451,A -85,B 0,C 180,E1 -28229.265,E2 -28229.265} C_VEL
LIN {X 0,Y 114.759,Z 428.025,A -85,B 0,C 180,E1 -28230.041,E2 -28230.041} C_VEL
LIN {X 0,Y 117.008,Z 403.811,A -85,B 0,C 180,E1 -28231.035,E2 -28231.035} C_VEL
LIN {X 0,Y 114.443,Z 394.852,A -85,B 0,C 180,E1 -28234.051,E2 -28234.051} C_VEL
LIN {X 0,Y 111.393,Z 388.563,A -85,B 0,C 180,E1 -28237.633,E2 -28237.633} C_VEL
LIN {X 0,Y 108.537,Z 383.317,A -85,B 0,C 180,E1 -28241.526,E2 -28241.526} C_VEL
LIN {X 0,Y 106.47,Z 379.779,A -85,B 0,C 180,E1 -28244.873,E2 -28244.873} C_VEL
LIN {X 0,Y 104.26,Z 375.974,A -85,B 0,C 180,E1 -28249.378,E2 -28249.378} C_VEL
LIN {X 0,Y 102.267,Z 372.406,A -85,B 0,C 180,E1 -28255.318,E2 -28255.318} C_VEL
LIN {X 0,Y 101.965,Z 371.59,A -85,B 0,C 180,E1 -28256.718,E2 -28256.718} C_VEL
LIN {X 0,Y 101.246,Z 371.732,A -85,B 0,C 180,E1 -28260.03,E2 -28260.03} C_VEL
LIN {X 0,Y 100.751,Z 372.849,A -85,B 0,C 180,E1 -28263.331,E2 -28263.331} C_VEL
LIN {X 0,Y 100.517,Z 376.754,A -85,B 0,C 180,E1 -28269.821,E2 -28269.821} C_VEL
LIN {X 0,Y 101.025,Z 379.627,A -85,B 0,C 180,E1 -28274.109,E2 -28274.109} C_VEL
LIN {X 0,Y 103.245,Z 383.617,A -85,B 0,C 180,E1 -28281.152,E2 -28281.152} C_VEL
LIN {X 0,Y 105.471,Z 387.751,A -85,B 0,C 180,E1 -28285.797,E2 -28285.797} C_VEL
LIN {X 0,Y 107.977,Z 392.374,A -85,B 0,C 180,E1 -28289.859,E2 -28289.859} C_VEL
LIN {X 0,Y 111.289,Z 399.483,A -85,B 0,C 180,E1 -28294.332,E2 -28294.332} C_VEL
LIN {X 0,Y 113.108,Z 403.789,A -85,B 0,C 180,E1 -28296.499,E2 -28296.499} C_VEL
LIN {X 0,Y 110.094,Z 433.976,A -85,B 0,C 180,E1 -28297.874,E2 -28297.874} C_VEL
LIN {X 0,Y 107.664,Z 447.26,A -85,B 0,C 180,E1 -28298.997,E2 -28298.997} C_VEL
LIN {X 0,Y 104.483,Z 459.029,A -85,B 0,C 180,E1 -28300.456,E2 -28300.456} C_VEL
LIN {X 0,Y 100.082,Z 471.023,A -85,B 0,C 180,E1 -28302.498,E2 -28302.498} C_VEL
LIN {X 0,Y 94.72,Z 482.503,A -85,B 0,C 180,E1 -28305.183,E2 -28305.183} C_VEL
LIN {X 0,Y 89.152,Z 492.806,A -85,B 0,C 180,E1 -28308.686,E2 -28308.686} C_VEL
LIN {X 0,Y 83.838,Z 501.247,A -85,B 0,C 180,E1 -28312.575,E2 -28312.575} C_VEL
LIN {X 0,Y 77.491,Z 510.376,A -85,B 0,C 180,E1 -28318.57,E2 -28318.57} C_VEL
LIN {X 0,Y 72.088,Z 517.727,A -85,B 0,C 180,E1 -28325.525,E2 -28325.525} C_VEL
LIN {X 0,Y 68.412,Z 522.72,A -85,B 0,C 180,E1 -28332.052,E2 -28332.052} C_VEL
LIN {X 0,Y 65.163,Z 527.571,A -85,B 0,C 180,E1 -28340.692,E2 -28340.692} C_VEL
LIN {X 0,Y 63.255,Z 531.535,A -85,B 0,C 180,E1 -28350.666,E2 -28350.666} C_VEL
LIN {X 0,Y 62.487,Z 534.794,A -85,B 0,C 180,E1 -28363.002,E2 -28363.002} C_VEL
LIN {X 0,Y 64.517,Z 536.549,A -85,B 0,C 180,E1 -28375.834,E2 -28375.834} C_VEL
LIN {X 0,Y 66.929,Z 536.852,A -85,B 0,C 180,E1 -28382.857,E2 -28382.857} C_VEL
LIN {X 0,Y 72.374,Z 536.152,A -85,B 0,C 180,E1 -28392.826,E2 -28392.826} C_VEL
LIN {X 0,Y 76.139,Z 535.197,A -85,B 0,C 180,E1 -28397.601,E2 -28397.601} C_VEL
LIN {X 0,Y 81.241,Z 533.489,A -85,B 0,C 180,E1 -28402.732,E2 -28402.732} C_VEL
LIN {X 0,Y 89.914,Z 529.69,A -85,B 0,C 180,E1 -28409.296,E2 -28409.296} C_VEL
LIN {X 0,Y 97.88,Z 525.314,A -85,B 0,C 180,E1 -28413.837,E2 -28413.837} C_VEL
LIN {X 0,Y 106.376,Z 519.698,A -85,B 0,C 180,E1 -28417.662,E2 -28417.662} C_VEL
LIN {X 0,Y 115.265,Z 512.627,A -85,B 0,C 180,E1 -28420.924,E2 -28420.924} C_VEL
LIN {X 0,Y 124.478,Z 503.714,A -85,B 0,C 180,E1 -28423.704,E2 -28423.704} C_VEL
LIN {X 0,Y 132.327,Z 494.532,A -85,B 0,C 180,E1 -28425.762,E2 -28425.762} C_VEL
LIN {X 0,Y 139.486,Z 484.306,A -85,B 0,C 180,E1 -28427.479,E2 -28427.479} C_VEL
LIN {X 0,Y 146.158,Z 472.5,A -85,B 0,C 180,E1 -28428.854,E2 -28428.854} C_VEL
LIN {X 0,Y 151.481,Z 460.414,A -85,B 0,C 180,E1 -28429.914,E2 -28429.914} C_VEL
LIN {X 0,Y 155.56,Z 447.742,A -85,B 0,C 180,E1 -28430.721,E2 -28430.721} C_VEL
LIN {X 0,Y 157.1,Z 441.385,A -85,B 0,C 180,E1 -28431.038,E2 -28431.038} C_VEL
LIN {X 0,Y 156.167,Z 437.851,A -85,B 0,C 180,E1 -28434.027,E2 -28434.027} C_VEL
LIN {X 0,Y 155.433,Z 435.364,A -85,B 0,C 180,E1 -28436.76,E2 -28436.76} C_VEL
LIN {X 0,Y 154.862,Z 433.065,A -85,B 0,C 180,E1 -28440.001,E2 -28440.001} C_VEL
LIN {X 0,Y 154.52,Z 432.446,A -85,B 0,C 180,E1 -28442.607,E2 -28442.607} C_VEL
LIN {X 0,Y 154.67,Z 433.063,A -85,B 0,C 180,E1 -28448.493,E2 -28448.493} C_VEL
LIN {X 0,Y 154.943,Z 433.664,A -85,B 0,C 180,E1 -28450.124,E2 -28450.124} C_VEL
LIN {X 0,Y 156.032,Z 437.176,A -85,B 0,C 180,E1 -28454.677,E2 -28454.677} C_VEL
LIN {X 0,Y 156.772,Z 440.978,A -85,B 0,C 180,E1 -28457.362,E2 -28457.362} C_VEL
LIN {X 0,Y 157.056,Z 443.261,A -85,B 0,C 180,E1 -28458.617,E2 -28458.617} C_VEL
LIN {X 0,Y 153.323,Z 457.085,A -85,B 0,C 180,E1 -28459.236,E2 -28459.236} C_VEL
LIN {X 0,Y 148.623,Z 469.224,A -85,B 0,C 180,E1 -28459.975,E2 -28459.975} C_VEL
LIN {X 0,Y 142.943,Z 480.474,A -85,B 0,C 180,E1 -28460.906,E2 -28460.906} C_VEL
LIN {X 0,Y 136.531,Z 490.761,A -85,B 0,C 180,E1 -28462.094,E2 -28462.094} C_VEL
LIN {X 0,Y 128.675,Z 501.168,A -85,B 0,C 180,E1 -28463.813,E2 -28463.813} C_VEL
LIN {X 0,Y 120.949,Z 509.613,A -85,B 0,C 180,E1 -28465.754,E2 -28465.754} C_VEL
LIN {X 0,Y 111.914,Z 517.869,A -85,B 0,C 180,E1 -28468.455,E2 -28468.455} C_VEL
LIN {X 0,Y 103.195,Z 524.543,A -85,B 0,C 180,E1 -28471.645,E2 -28471.645} C_VEL
LIN {X 0,Y 94.906,Z 529.894,A -85,B 0,C 180,E1 -28475.453,E2 -28475.453} C_VEL
LIN {X 0,Y 86.288,Z 534.559,A -85,B 0,C 180,E1 -28480.663,E2 -28480.663} C_VEL
LIN {X 0,Y 80.264,Z 537.254,A -85,B 0,C 180,E1 -28485.532,E2 -28485.532} C_VEL
LIN {X 0,Y 75.991,Z 538.845,A -85,B 0,C 180,E1 -28489.653,E2 -28489.653} C_VEL
LIN {X 0,Y 72.242,Z 540.024,A -85,B 0,C 180,E1 -28494.286,E2 -28494.286} C_VEL
LIN {X 0,Y 66.418,Z 541.168,A -85,B 0,C 180,E1 -28504.957,E2 -28504.957} C_VEL
LIN {X 0,Y 63.259,Z 540.805,A -85,B 0,C 180,E1 -28517.16,E2 -28517.16} C_VEL
LIN {X 0,Y 62.723,Z 540.005,A -85,B 0,C 180,E1 -28523.564,E2 -28523.564} C_VEL
LIN {X 0,Y 62.789,Z 538.803,A -85,B 0,C 180,E1 -28529.998,E2 -28529.998} C_VEL
LIN {X 0,Y 62.882,Z 536.143,A -85,B 0,C 180,E1 -28539.649,E2 -28539.649} C_VEL
LIN {X 0,Y 64.37,Z 532.433,A -85,B 0,C 180,E1 -28549.117,E2 -28549.117} C_VEL
LIN {X 0,Y 67.352,Z 527.581,A -85,B 0,C 180,E1 -28558.003,E2 -28558.003} C_VEL
LIN {X 0,Y 71.779,Z 521.447,A -85,B 0,C 180,E1 -28565.975,E2 -28565.975} C_VEL
LIN {X 0,Y 76.362,Z 515.093,A -85,B 0,C 180,E1 -28571.948,E2 -28571.948} C_VEL
LIN {X 0,Y 82.724,Z 505.966,A -85,B 0,C 180,E1 -28578.017,E2 -28578.017} C_VEL
LIN {X 0,Y 89.323,Z 495.305,A -85,B 0,C 180,E1 -28582.808,E2 -28582.808} C_VEL
LIN {X 0,Y 95.219,Z 484.465,A -85,B 0,C 180,E1 -28586.131,E2 -28586.131} C_VEL
LIN {X 0,Y 99.965,Z 473.889,A -85,B 0,C 180,E1 -28588.475,E2 -28588.475} C_VEL
LIN {X 0,Y 104.536,Z 461.137,A -85,B 0,C 180,E1 -28590.431,E2 -28590.431} C_VEL
LIN {X 0,Y 107.905,Z 448.36,A -85,B 0,C 180,E1 -28591.792,E2 -28591.792} C_VEL
LIN {X 0,Y 110.084,Z 435.377,A -85,B 0,C 180,E1 -28592.7,E2 -28592.7} C_VEL
LIN {X 0,Y 112.979,Z 405.945,A -85,B 0,C 180,E1 -28593.938,E2 -28593.938} C_VEL
LIN {X 0,Y 111.197,Z 399.346,A -85,B 0,C 180,E1 -28596.362,E2 -28596.362} C_VEL
LIN {X 0,Y 108.122,Z 392.559,A -85,B 0,C 180,E1 -28600.54,E2 -28600.54} C_VEL
LIN {X 0,Y 105.74,Z 388.158,A -85,B 0,C 180,E1 -28604.334,E2 -28604.334} C_VEL
LIN {X 0,Y 104.521,Z 385.914,A -85,B 0,C 180,E1 -28606.635,E2 -28606.635} C_VEL
LIN {X 0,Y 102.791,Z 382.557,A -85,B 0,C 180,E1 -28610.654,E2 -28610.654} C_VEL
LIN {X 0,Y 100.849,Z 378.488,A -85,B 0,C 180,E1 -28617.753,E2 -28617.753} C_VEL
LIN {X 0,Y 100.457,Z 378.114,A -85,B 0,C 180,E1 -28619.999,E2 -28619.999} C_VEL
LIN {X 0,Y 100.348,Z 378.392,A -85,B 0,C 180,E1 -28630.083,E2 -28630.083} C_VEL
LIN {X 0,Y 100.835,Z 378.88,A -85,B 0,C 180,E1 -28632.986,E2 -28632.986} C_VEL
LIN {X 0,Y 101.025,Z 379.627,A -85,B 0,C 180,E1 -28634.109,E2 -28634.109} C_VEL
LIN {X 0,Y 101.669,Z 382.151,A -85,B 0,C 180,E1 -28637.122,E2 -28637.122} C_VEL
LIN {X 0,Y 102.383,Z 385.485,A -85,B 0,C 180,E1 -28639.866,E2 -28639.866} C_VEL
LIN {X 0,Y 105.779,Z 398.392,A -85,B 0,C 180,E1 -28648.159,E2 -28648.159} C_VEL
LIN {X 0,Y 108.566,Z 404.889,A -85,B 0,C 180,E1 -28652.391,E2 -28652.391} C_VEL
LIN {X 0,Y 109.305,Z 406.771,A -85,B 0,C 180,E1 -28653.403,E2 -28653.403} C_VEL
LIN {X 0,Y 106.402,Z 434.519,A -85,B 0,C 180,E1 -28654.671,E2 -28654.671} C_VEL
LIN {X 0,Y 103.735,Z 448.272,A -85,B 0,C 180,E1 -28655.821,E2 -28655.821} C_VEL
LIN {X 0,Y 100.394,Z 459.83,A -85,B 0,C 180,E1 -28657.225,E2 -28657.225} C_VEL
LIN {X 0,Y 96.152,Z 470.886,A -85,B 0,C 180,E1 -28659.052,E2 -28659.052} C_VEL
LIN {X 0,Y 90.517,Z 482.44,A -85,B 0,C 180,E1 -28661.645,E2 -28661.645} C_VEL
LIN {X 0,Y 84.61,Z 492.801,A -85,B 0,C 180,E1 -28665.089,E2 -28665.089} C_VEL
LIN {X 0,Y 78.33,Z 502.136,A -85,B 0,C 180,E1 -28669.425,E2 -28669.425} C_VEL
LIN {X 0,Y 71.536,Z 511.147,A -85,B 0,C 180,E1 -28675.607,E2 -28675.607} C_VEL
LIN {X 0,Y 65.697,Z 518.409,A -85,B 0,C 180,E1 -28682.96,E2 -28682.96} C_VEL
LIN {X 0,Y 61.68,Z 523.324,A -85,B 0,C 180,E1 -28690.014,E2 -28690.014} C_VEL
LIN {X 0,Y 58.178,Z 528.102,A -85,B 0,C 180,E1 -28699.563,E2 -28699.563} C_VEL
LIN {X 0,Y 56.184,Z 531.778,A -85,B 0,C 180,E1 -28710.003,E2 -28710.003} C_VEL
LIN {X 0,Y 55.421,Z 533.707,A -85,B 0,C 180,E1 -28717.288,E2 -28717.288} C_VEL
LIN {X 0,Y 55.463,Z 535.17,A -85,B 0,C 180,E1 -28724.683,E2 -28724.683} C_VEL
LIN {X 0,Y 58.061,Z 536.866,A -85,B 0,C 180,E1 -28738.961,E2 -28738.961} C_VEL
LIN {X 0,Y 60.56,Z 537.122,A -85,B 0,C 180,E1 -28745.677,E2 -28745.677} C_VEL
LIN {X 0,Y 67.203,Z 536.348,A -85,B 0,C 180,E1 -28757.061,E2 -28757.061} C_VEL
LIN {X 0,Y 71.432,Z 535.361,A -85,B 0,C 180,E1 -28761.918,E2 -28761.918} C_VEL
LIN {X 0,Y 76.316,Z 533.857,A -85,B 0,C 180,E1 -28766.46,E2 -28766.46} C_VEL
LIN {X 0,Y 83.707,Z 530.975,A -85,B 0,C 180,E1 -28771.836,E2 -28771.836} C_VEL
LIN {X 0,Y 92.011,Z 526.912,A -85,B 0,C 180,E1 -28776.435,E2 -28776.435} C_VEL
LIN {X 0,Y 102.31,Z 520.614,A -85,B 0,C 180,E1 -28780.829,E2 -28780.829} C_VEL
LIN {X 0,Y 111.537,Z 513.716,A -85,B 0,C 180,E1 -28783.93,E2 -28783.93} C_VEL
LIN {X 0,Y 120.078,Z 506.028,A -85,B 0,C 180,E1 -28786.295,E2 -28786.295} C_VEL
LIN {X 0,Y 127.481,Z 498.045,A -85,B 0,C 180,E1 -28788.114,E2 -28788.114} C_VEL
LIN {X 0,Y 135.623,Z 487.345,A -85,B 0,C 180,E1 -28789.929,E2 -28789.929} C_VEL
LIN {X 0,Y 142.247,Z 476.7,A -85,B 0,C 180,E1 -28791.171,E2 -28791.171} C_VEL
LIN {X 0,Y 147.398,Z 466.355,A -85,B 0,C 180,E1 -28792.128,E2 -28792.128} C_VEL
LIN {X 0,Y 151.887,Z 454.844,A -85,B 0,C 180,E1 -28792.902,E2 -28792.902} C_VEL
LIN {X 0,Y 154.491,Z 445.966,A -85,B 0,C 180,E1 -28793.387,E2 -28793.387} C_VEL
LIN {X 0,Y 154.062,Z 443.417,A -85,B 0,C 180,E1 -28795.749,E2 -28795.749} C_VEL
LIN {X 0,Y 153.522,Z 440.075,A -85,B 0,C 180,E1 -28800.001,E2 -28800.001} C_VEL
LIN {X 0,Y 153.25,Z 439.439,A -85,B 0,C 180,E1 -28802.629,E2 -28802.629} C_VEL
LIN {X 0,Y 153.406,Z 440.086,A -85,B 0,C 180,E1 -28808.563,E2 -28808.563} C_VEL
LIN {X 0,Y 153.555,Z 440.758,A -85,B 0,C 180,E1 -28809.883,E2 -28809.883} C_VEL
LIN {X 0,Y 154.278,Z 443.823,A -85,B 0,C 180,E1 -28814.006,E2 -28814.006} C_VEL
LIN {X 0,Y 154.613,Z 446.891,A -85,B 0,C 180,E1 -28816.166,E2 -28816.166} C_VEL
LIN {X 0,Y 150.762,Z 459.527,A -85,B 0,C 180,E1 -28816.764,E2 -28816.764} C_VEL
LIN {X 0,Y 145.535,Z 471.938,A -85,B 0,C 180,E1 -28817.494,E2 -28817.494} C_VEL
LIN {X 0,Y 139.766,Z 482.614,A -85,B 0,C 180,E1 -28818.355,E2 -28818.355} C_VEL
LIN {X 0,Y 134.038,Z 491.308,A -85,B 0,C 180,E1 -28819.3,E2 -28819.3} C_VEL
LIN {X 0,Y 125.984,Z 501.532,A -85,B 0,C 180,E1 -28820.867,E2 -28820.867} C_VEL
LIN {X 0,Y 118.043,Z 509.864,A -85,B 0,C 180,E1 -28822.655,E2 -28822.655} C_VEL
LIN {X 0,Y 108.716,Z 518.031,A -85,B 0,C 180,E1 -28825.169,E2 -28825.169} C_VEL
LIN {X 0,Y 99.651,Z 524.628,A -85,B 0,C 180,E1 -28828.165,E2 -28828.165} C_VEL
LIN {X 0,Y 90.967,Z 529.907,A -85,B 0,C 180,E1 -28831.803,E2 -28831.803} C_VEL
LIN {X 0,Y 81.083,Z 534.804,A -85,B 0,C 180,E1 -28837.355,E2 -28837.355} C_VEL
LIN {X 0,Y 75.337,Z 537.139,A -85,B 0,C 180,E1 -28841.727,E2 -28841.727} C_VEL
LIN {X 0,Y 70.712,Z 538.7,A -85,B 0,C 180,E1 -28845.913,E2 -28845.913} C_VEL
LIN {X 0,Y 62.944,Z 540.556,A -85,B 0,C 180,E1 -28856.061,E2 -28856.061} C_VEL
LIN {X 0,Y 57.827,Z 540.9,A -85,B 0,C 180,E1 -28868.614,E2 -28868.614} C_VEL
LIN {X 0,Y 56.335,Z 540.48,A -85,B 0,C 180,E1 -28875.549,E2 -28875.549} C_VEL
LIN {X 0,Y 55.657,Z 539.646,A -85,B 0,C 180,E1 -28882.743,E2 -28882.743} C_VEL
LIN {X 0,Y 55.685,Z 538.417,A -85,B 0,C 180,E1 -28889.997,E2 -28889.997} C_VEL
LIN {X 0,Y 55.878,Z 535.7,A -85,B 0,C 180,E1 -28900.872,E2 -28900.872} C_VEL
LIN {X 0,Y 57.651,Z 531.927,A -85,B 0,C 180,E1 -28911.449,E2 -28911.449} C_VEL
LIN {X 0,Y 61.134,Z 527.012,A -85,B 0,C 180,E1 -28921.15,E2 -28921.15} C_VEL
LIN {X 0,Y 66.108,Z 520.804,A -85,B 0,C 180,E1 -28929.629,E2 -28929.629} C_VEL
LIN {X 0,Y 70.881,Z 514.761,A -85,B 0,C 180,E1 -28935.487,E2 -28935.487} C_VEL
LIN {X 0,Y 76.908,Z 506.809,A -85,B 0,C 180,E1 -28940.96,E2 -28940.96} C_VEL
LIN {X 0,Y 83.22,Z 497.547,A -85,B 0,C 180,E1 -28945.422,E2 -28945.422} C_VEL
LIN {X 0,Y 89.305,Z 487.234,A -85,B 0,C 180,E1 -28948.847,E2 -28948.847} C_VEL
LIN {X 0,Y 94.98,Z 475.787,A -85,B 0,C 180,E1 -28951.48,E2 -28951.48} C_VEL
LIN {X 0,Y 99.734,Z 463.875,A -85,B 0,C 180,E1 -28953.383,E2 -28953.383} C_VEL
LIN {X 0,Y 103.458,Z 451.202,A -85,B 0,C 180,E1 -28954.804,E2 -28954.804} C_VEL
LIN {X 0,Y 106.189,Z 437.3,A -85,B 0,C 180,E1 -28955.826,E2 -28955.826} C_VEL
LIN {X 0,Y 109.251,Z 408.167,A -85,B 0,C 180,E1 -28957.046,E2 -28957.046} C_VEL
LIN {X 0,Y 108.178,Z 403.942,A -85,B 0,C 180,E1 -28958.752,E2 -28958.752} C_VEL
LIN {X 0,Y 105.633,Z 397.961,A -85,B 0,C 180,E1 -28962.703,E2 -28962.703} C_VEL
LIN {X 0,Y 103.144,Z 392.754,A -85,B 0,C 180,E1 -28967.455,E2 -28967.455} C_VEL
LIN {X 0,Y 101.348,Z 389.154,A -85,B 0,C 180,E1 -28972.027,E2 -28972.027} C_VEL
LIN {X 0,Y 99.826,Z 385.423,A -85,B 0,C 180,E1 -28978.486,E2 -28978.486} C_VEL
LIN {X 0,Y 99.203,Z 385.077,A -85,B 0,C 180,E1 -28984.062,E2 -28984.062} C_VEL
LIN {X 0,Y 99.762,Z 385.683,A -85,B 0,C 180,E1 -28991.942,E2 -28991.942} C_VEL
LIN {X 0,Y 101.194,Z 389.23,A -85,B 0,C 180,E1 -28998.211,E2 -28998.211} C_VEL
LIN {X 0,Y 101.885,Z 390.513,A -85,B 0,C 180,E1 -29000.175,E2 -29000.175} C_VEL
LIN {X 0,Y 103.7,Z 394.137,A -85,B 0,C 180,E1 -29004.368,E2 -29004.368} C_VEL
LIN {X 0,Y 105.779,Z 398.392,A -85,B 0,C 180,E1 -29008.159,E2 -29008.159} C_VEL
LIN {X 0,Y 106.466,Z 401.205,A -85,B 0,C 180,E1 -29009.476,E2 -29009.476} C_VEL
LIN {X 0,Y 106.729,Z 404.694,A -85,B 0,C 180,E1 -29010.32,E2 -29010.32} C_VEL
LIN {X 0,Y 106.497,Z 410.528,A -85,B 0,C 180,E1 -29010.925,E2 -29010.925} C_VEL
LIN {X 0,Y 103.786,Z 429.771,A -85,B 0,C 180,E1 -29010.979,E2 -29010.979} C_VEL
LIN {X 0,Y 101.565,Z 443.175,A -85,B 0,C 180,E1 -29011.845,E2 -29011.845} C_VEL
LIN {X 0,Y 98.156,Z 456.117,A -85,B 0,C 180,E1 -29013.197,E2 -29013.197} C_VEL
LIN {X 0,Y 93.359,Z 468.996,A -85,B 0,C 180,E1 -29015.052,E2 -29015.052} C_VEL
LIN {X 0,Y 88.127,Z 479.742,A -85,B 0,C 180,E1 -29017.113,E2 -29017.113} C_VEL
LIN {X 0,Y 81.809,Z 490.64,A -85,B 0,C 180,E1 -29020.324,E2 -29020.324} C_VEL
LIN {X 0,Y 75.704,Z 499.531,A -85,B 0,C 180,E1 -29023.992,E2 -29023.992} C_VEL
LIN {X 0,Y 68.151,Z 509.176,A -85,B 0,C 180,E1 -29029.873,E2 -29029.873} C_VEL
LIN {X 0,Y 61.496,Z 516.847,A -85,B 0,C 180,E1 -29037.126,E2 -29037.126} C_VEL
LIN {X 0,Y 55.047,Z 523.924,A -85,B 0,C 180,E1 -29047.482,E2 -29047.482} C_VEL
LIN {X 0,Y 51.22,Z 528.628,A -85,B 0,C 180,E1 -29058.126,E2 -29058.126} C_VEL
LIN {X 0,Y 48.998,Z 532.244,A -85,B 0,C 180,E1 -29070.003,E2 -29070.003} C_VEL
LIN {X 0,Y 48.291,Z 534.128,A -85,B 0,C 180,E1 -29078.371,E2 -29078.371} C_VEL
LIN {X 0,Y 48.511,Z 535.544,A -85,B 0,C 180,E1 -29086.846,E2 -29086.846} C_VEL
LIN {X 0,Y 49.721,Z 536.558,A -85,B 0,C 180,E1 -29095.093,E2 -29095.093} C_VEL
LIN {X 0,Y 54.331,Z 537.387,A -85,B 0,C 180,E1 -29109.095,E2 -29109.095} C_VEL
LIN {X 0,Y 58.301,Z 537.161,A -85,B 0,C 180,E1 -29116.329,E2 -29116.329} C_VEL
LIN {X 0,Y 62.462,Z 536.545,A -85,B 0,C 180,E1 -29121.966,E2 -29121.966} C_VEL
LIN {X 0,Y 67.176,Z 535.529,A -85,B 0,C 180,E1 -29126.824,E2 -29126.824} C_VEL
LIN {X 0,Y 72.274,Z 534.053,A -85,B 0,C 180,E1 -29131.068,E2 -29131.068} C_VEL
LIN {X 0,Y 80.532,Z 531.017,A -85,B 0,C 180,E1 -29136.398,E2 -29136.398} C_VEL
LIN {X 0,Y 89.355,Z 526.885,A -85,B 0,C 180,E1 -29140.709,E2 -29140.709} C_VEL
LIN {X 0,Y 100.157,Z 520.513,A -85,B 0,C 180,E1 -29144.764,E2 -29144.764} C_VEL
LIN {X 0,Y 109.751,Z 513.528,A -85,B 0,C 180,E1 -29147.571,E2 -29147.571} C_VEL
LIN {X 0,Y 119.489,Z 504.772,A -85,B 0,C 180,E1 -29149.93,E2 -29149.93} C_VEL
LIN {X 0,Y 128.682,Z 494.621,A -85,B 0,C 180,E1 -29151.853,E2 -29151.853} C_VEL
LIN {X 0,Y 136.23,Z 484.254,A -85,B 0,C 180,E1 -29153.267,E2 -29153.267} C_VEL
LIN {X 0,Y 143.084,Z 472.558,A -85,B 0,C 180,E1 -29154.363,E2 -29154.363} C_VEL
LIN {X 0,Y 148.117,Z 461.607,A -85,B 0,C 180,E1 -29155.162,E2 -29155.162} C_VEL
LIN {X 0,Y 151.492,Z 452.144,A -85,B 0,C 180,E1 -29155.706,E2 -29155.706} C_VEL
LIN {X 0,Y 151.983,Z 450.33,A -85,B 0,C 180,E1 -29156.022,E2 -29156.022} C_VEL
LIN {X 0,Y 151.713,Z 447.816,A -85,B 0,C 180,E1 -29159.171,E2 -29159.171} C_VEL
LIN {X 0,Y 151.692,Z 446.79,A -85,B 0,C 180,E1 -29160.664,E2 -29160.664} C_VEL
LIN {X 0,Y 151.565,Z 446.322,A -85,B 0,C 180,E1 -29162.658,E2 -29162.658} C_VEL
LIN {X 0,Y 151.648,Z 446.841,A -85,B 0,C 180,E1 -29167.992,E2 -29167.992} C_VEL
LIN {X 0,Y 151.753,Z 447.833,A -85,B 0,C 180,E1 -29169.834,E2 -29169.834} C_VEL
LIN {X 0,Y 152.178,Z 450.349,A -85,B 0,C 180,E1 -29173.267,E2 -29173.267} C_VEL
LIN {X 0,Y 152.133,Z 451.228,A -85,B 0,C 180,E1 -29173.76,E2 -29173.76} C_VEL
LIN {X 0,Y 147.636,Z 463.969,A -85,B 0,C 180,E1 -29174.318,E2 -29174.318} C_VEL
LIN {X 0,Y 141.889,Z 476.05,A -85,B 0,C 180,E1 -29175.011,E2 -29175.011} C_VEL
LIN {X 0,Y 135.179,Z 487.15,A -85,B 0,C 180,E1 -29175.882,E2 -29175.882} C_VEL
LIN {X 0,Y 126.925,Z 498.107,A -85,B 0,C 180,E1 -29177.222,E2 -29177.222} C_VEL
LIN {X 0,Y 118.7,Z 507.011,A -85,B 0,C 180,E1 -29178.677,E2 -29178.677} C_VEL
LIN {X 0,Y 109.076,Z 515.718,A -85,B 0,C 180,E1 -29180.887,E2 -29180.887} C_VEL
LIN {X 0,Y 99.601,Z 522.694,A -85,B 0,C 180,E1 -29183.463,E2 -29183.463} C_VEL
LIN {X 0,Y 90.402,Z 528.301,A -85,B 0,C 180,E1 -29186.614,E2 -29186.614} C_VEL
LIN {X 0,Y 81.625,Z 532.736,A -85,B 0,C 180,E1 -29190.567,E2 -29190.567} C_VEL
LIN {X 0,Y 76.044,Z 535.091,A -85,B 0,C 180,E1 -29193.715,E2 -29193.715} C_VEL
LIN {X 0,Y 70.79,Z 537.029,A -85,B 0,C 180,E1 -29197.415,E2 -29197.415} C_VEL
LIN {X 0,Y 65.783,Z 538.545,A -85,B 0,C 180,E1 -29201.593,E2 -29201.593} C_VEL
LIN {X 0,Y 57.178,Z 540.333,A -85,B 0,C 180,E1 -29212.077,E2 -29212.077} C_VEL
LIN {X 0,Y 51.255,Z 540.617,A -85,B 0,C 180,E1 -29225.707,E2 -29225.707} C_VEL
LIN {X 0,Y 48.608,Z 539.287,A -85,B 0,C 180,E1 -29241.684,E2 -29241.684} C_VEL
LIN {X 0,Y 48.58,Z 538.032,A -85,B 0,C 180,E1 -29249.997,E2 -29249.997} C_VEL
LIN {X 0,Y 48.92,Z 535.257,A -85,B 0,C 180,E1 -29262.442,E2 -29262.442} C_VEL
LIN {X 0,Y 51.065,Z 531.422,A -85,B 0,C 180,E1 -29274.383,E2 -29274.383} C_VEL
LIN {X 0,Y 55.15,Z 526.443,A -85,B 0,C 180,E1 -29284.988,E2 -29284.988} C_VEL
LIN {X 0,Y 60.772,Z 520.163,A -85,B 0,C 180,E1 -29293.934,E2 -29293.934} C_VEL
LIN {X 0,Y 65.168,Z 515.094,A -85,B 0,C 180,E1 -29299.014,E2 -29299.014} C_VEL
LIN {X 0,Y 72.609,Z 505.99,A -85,B 0,C 180,E1 -29305.356,E2 -29305.356} C_VEL
LIN {X 0,Y 79.389,Z 496.577,A -85,B 0,C 180,E1 -29309.665,E2 -29309.665} C_VEL
LIN {X 0,Y 85.85,Z 486.097,A -85,B 0,C 180,E1 -29312.902,E2 -29312.902} C_VEL
LIN {X 0,Y 91.037,Z 476.04,A -85,B 0,C 180,E1 -29315.102,E2 -29315.102} C_VEL
LIN {X 0,Y 95.987,Z 464.265,A -85,B 0,C 180,E1 -29316.892,E2 -29316.892} C_VEL
LIN {X 0,Y 99.894,Z 451.793,A -85,B 0,C 180,E1 -29318.238,E2 -29318.238} C_VEL
LIN {X 0,Y 102.7,Z 438.463,A -85,B 0,C 180,E1 -29319.199,E2 -29319.199} C_VEL
LIN {X 0,Y 105.848,Z 410.431,A -85,B 0,C 180,E1 -29320.358,E2 -29320.358} C_VEL
LIN {X 0,Y 104.902,Z 407.361,A -85,B 0,C 180,E1 -29322.019,E2 -29322.019} C_VEL
LIN {X 0,Y 102.617,Z 401.698,A -85,B 0,C 180,E1 -29326.382,E2 -29326.382} C_VEL
LIN {X 0,Y 100.992,Z 398.186,A -85,B 0,C 180,E1 -29330.233,E2 -29330.233} C_VEL
LIN {X 0,Y 99.996,Z 395.762,A -85,B 0,C 180,E1 -29333.349,E2 -29333.349} C_VEL
LIN {X 0,Y 98.858,Z 392.428,A -85,B 0,C 180,E1 -29338.981,E2 -29338.981} C_VEL
LIN {X 0,Y 98.311,Z 392.24,A -85,B 0,C 180,E1 -29346.155,E2 -29346.155} C_VEL
LIN {X 0,Y 98.759,Z 392.753,A -85,B 0,C 180,E1 -29351.285,E2 -29351.285} C_VEL
LIN {X 0,Y 100.394,Z 396.87,A -85,B 0,C 180,E1 -29358.625,E2 -29358.625} C_VEL
LIN {X 0,Y 102.068,Z 400.675,A -85,B 0,C 180,E1 -29363.054,E2 -29363.054} C_VEL
LIN {X 0,Y 103.878,Z 404.893,A -85,B 0,C 180,E1 -29366.764,E2 -29366.764} C_VEL
LIN {X 0,Y 105.836,Z 409.895,A -85,B 0,C 180,E1 -29370.139,E2 -29370.139} C_VEL
LIN {X 0,Y 103.786,Z 429.771,A -85,B 0,C 180,E1 -29370.979,E2 -29370.979} C_VEL
LIN {X 0,Y 102.715,Z 435.577,A -85,B 0,C 180,E1 -29370.976,E2 -29370.976} C_VEL
LIN {X 0,Y 99.682,Z 444.915,A -85,B 0,C 180,E1 -29370.196,E2 -29370.196} C_VEL
LIN {X 0,Y 96.021,Z 454.099,A -85,B 0,C 180,E1 -29369.526,E2 -29369.526} C_VEL
LIN {X 0,Y 93.915,Z 459.597,A -85,B 0,C 180,E1 -29369.778,E2 -29369.778} C_VEL
LIN {X 0,Y 89.465,Z 470.524,A -85,B 0,C 180,E1 -29371.323,E2 -29371.323} C_VEL
LIN {X 0,Y 84.043,Z 480.967,A -85,B 0,C 180,E1 -29373.259,E2 -29373.259} C_VEL
LIN {X 0,Y 77.432,Z 491.669,A -85,B 0,C 180,E1 -29376.342,E2 -29376.342} C_VEL
LIN {X 0,Y 69.571,Z 502.209,A -85,B 0,C 180,E1 -29380.747,E2 -29380.747} C_VEL
LIN {X 0,Y 61.63,Z 511.304,A -85,B 0,C 180,E1 -29386.83,E2 -29386.83} C_VEL
LIN {X 0,Y 54.536,Z 518.632,A -85,B 0,C 180,E1 -29394.559,E2 -29394.559} C_VEL
LIN {X 0,Y 48.552,Z 524.515,A -85,B 0,C 180,E1 -29404.266,E2 -29404.266} C_VEL
LIN {X 0,Y 44.303,Z 529.149,A -85,B 0,C 180,E1 -29416.238,E2 -29416.238} C_VEL
LIN {X 0,Y 41.806,Z 532.707,A -85,B 0,C 180,E1 -29430.003,E2 -29430.003} C_VEL
LIN {X 0,Y 41.154,Z 534.532,A -85,B 0,C 180,E1 -29439.836,E2 -29439.836} C_VEL
LIN {X 0,Y 41.664,Z 535.915,A -85,B 0,C 180,E1 -29449.72,E2 -29449.72} C_VEL
LIN {X 0,Y 43.283,Z 536.9,A -85,B 0,C 180,E1 -29459.155,E2 -29459.155} C_VEL
LIN {X 0,Y 48.313,Z 537.644,A -85,B 0,C 180,E1 -29473.339,E2 -29473.339} C_VEL
LIN {X 0,Y 53.528,Z 537.388,A -85,B 0,C 180,E1 -29481.981,E2 -29481.981} C_VEL
LIN {X 0,Y 58.251,Z 536.742,A -85,B 0,C 180,E1 -29487.628,E2 -29487.628} C_VEL
LIN {X 0,Y 67.698,Z 534.577,A -85,B 0,C 180,E1 -29495.466,E2 -29495.466} C_VEL
LIN {X 0,Y 77.895,Z 531.059,A -85,B 0,C 180,E1 -29501.33,E2 -29501.33} C_VEL
LIN {X 0,Y 87.218,Z 526.857,A -85,B 0,C 180,E1 -29505.234,E2 -29505.234} C_VEL
LIN {X 0,Y 98.495,Z 520.411,A -85,B 0,C 180,E1 -29508.854,E2 -29508.854} C_VEL
LIN {X 0,Y 108.423,Z 513.312,A -85,B 0,C 180,E1 -29511.31,E2 -29511.31} C_VEL
LIN {X 0,Y 117.797,Z 505.065,A -85,B 0,C 180,E1 -29513.27,E2 -29513.27} C_VEL
LIN {X 0,Y 127.001,Z 495.163,A -85,B 0,C 180,E1 -29514.935,E2 -29514.935} C_VEL
LIN {X 0,Y 134.71,Z 484.885,A -85,B 0,C 180,E1 -29516.184,E2 -29516.184} C_VEL
LIN {X 0,Y 141.764,Z 473.131,A -85,B 0,C 180,E1 -29517.159,E2 -29517.159} C_VEL
LIN {X 0,Y 146.989,Z 462.029,A -85,B 0,C 180,E1 -29517.876,E2 -29517.876} C_VEL
LIN {X 0,Y 149.499,Z 455.379,A -85,B 0,C 180,E1 -29518.316,E2 -29518.316} C_VEL
LIN {X 0,Y 149.489,Z 454.22,A -85,B 0,C 180,E1 -29520.001,E2 -29520.001} C_VEL
LIN {X 0,Y 149.491,Z 453.106,A -85,B 0,C 180,E1 -29522.695,E2 -29522.695} C_VEL
LIN {X 0,Y 149.579,Z 453.668,A -85,B 0,C 180,E1 -29528.104,E2 -29528.104} C_VEL
LIN {X 0,Y 149.643,Z 455.618,A -85,B 0,C 180,E1 -29531.056,E2 -29531.056} C_VEL
LIN {X 0,Y 149.485,Z 456.307,A -85,B 0,C 180,E1 -29531.295,E2 -29531.295} C_VEL
LIN {X 0,Y 144.236,Z 469.103,A -85,B 0,C 180,E1 -29531.827,E2 -29531.827} C_VEL
LIN {X 0,Y 137.673,Z 481.219,A -85,B 0,C 180,E1 -29532.496,E2 -29532.496} C_VEL
LIN {X 0,Y 130.893,Z 491.236,A -85,B 0,C 180,E1 -29533.297,E2 -29533.297} C_VEL
LIN {X 0,Y 123.33,Z 500.454,A -85,B 0,C 180,E1 -29534.36,E2 -29534.36} C_VEL
LIN {X 0,Y 114.98,Z 508.883,A -85,B 0,C 180,E1 -29535.697,E2 -29535.697} C_VEL
LIN {X 0,Y 105.118,Z 517.125,A -85,B 0,C 180,E1 -29537.684,E2 -29537.684} C_VEL
LIN {X 0,Y 95.38,Z 523.789,A -85,B 0,C 180,E1 -29540.034,E2 -29540.034} C_VEL
LIN {X 0,Y 84.345,Z 529.921,A -85,B 0,C 180,E1 -29543.568,E2 -29543.568} C_VEL
LIN {X 0,Y 75.259,Z 533.929,A -85,B 0,C 180,E1 -29547.48,E2 -29547.48} C_VEL
LIN {X 0,Y 66.699,Z 536.918,A -85,B 0,C 180,E1 -29552.544,E2 -29552.544} C_VEL
LIN {X 0,Y 61.289,Z 538.378,A -85,B 0,C 180,E1 -29556.609,E2 -29556.609} C_VEL
LIN {X 0,Y 51.753,Z 540.109,A -85,B 0,C 180,E1 -29567.232,E2 -29567.232} C_VEL
LIN {X 0,Y 47.871,Z 540.411,A -85,B 0,C 180,E1 -29574.035,E2 -29574.035} C_VEL
LIN {X 0,Y 44.842,Z 540.318,A -85,B 0,C 180,E1 -29581.95,E2 -29581.95} C_VEL
LIN {X 0,Y 41.597,Z 538.925,A -85,B 0,C 180,E1 -29600.27,E2 -29600.27} C_VEL
LIN {X 0,Y 41.469,Z 537.642,A -85,B 0,C 180,E1 -29609.997,E2 -29609.997} C_VEL
LIN {X 0,Y 41.995,Z 534.808,A -85,B 0,C 180,E1 -29624.535,E2 -29624.535} C_VEL
LIN {X 0,Y 44.659,Z 530.909,A -85,B 0,C 180,E1 -29638.168,E2 -29638.168} C_VEL
LIN {X 0,Y 49.471,Z 525.862,A -85,B 0,C 180,E1 -29649.734,E2 -29649.734} C_VEL
LIN {X 0,Y 55.853,Z 519.503,A -85,B 0,C 180,E1 -29659.019,E2 -29659.019} C_VEL
LIN {X 0,Y 63.045,Z 511.817,A -85,B 0,C 180,E1 -29666.124,E2 -29666.124} C_VEL
LIN {X 0,Y 70.198,Z 503.35,A -85,B 0,C 180,E1 -29671.161,E2 -29671.161} C_VEL
LIN {X 0,Y 77.478,Z 493.387,A -85,B 0,C 180,E1 -29675.101,E2 -29675.101} C_VEL
LIN {X 0,Y 83.578,Z 483.611,A -85,B 0,C 180,E1 -29677.66,E2 -29677.66} C_VEL
LIN {X 0,Y 89.025,Z 473.016,A -85,B 0,C 180,E1 -29679.623,E2 -29679.623} C_VEL
LIN {X 0,Y 93.795,Z 461.388,A -85,B 0,C 180,E1 -29681.075,E2 -29681.075} C_VEL
LIN {X 0,Y 97.882,Z 447.809,A -85,B 0,C 180,E1 -29682.261,E2 -29682.261} C_VEL
LIN {X 0,Y 100.31,Z 435.226,A -85,B 0,C 180,E1 -29683.012,E2 -29683.012} C_VEL
LIN {X 0,Y 102.771,Z 413.389,A -85,B 0,C 180,E1 -29683.804,E2 -29683.804} C_VEL
LIN {X 0,Y 100.894,Z 408.035,A -85,B 0,C 180,E1 -29687.937,E2 -29687.937} C_VEL
LIN {X 0,Y 99.544,Z 404.68,A -85,B 0,C 180,E1 -29691.626,E2 -29691.626} C_VEL
LIN {X 0,Y 98.678,Z 402.314,A -85,B 0,C 180,E1 -29694.795,E2 -29694.795} C_VEL
LIN {X 0,Y 97.831,Z 399.29,A -85,B 0,C 180,E1 -29699.999,E2 -29699.999} C_VEL
LIN {X 0,Y 97.542,Z 399.398,A -85,B 0,C 180,E1 -29708.284,E2 -29708.284} C_VEL
LIN {X 0,Y 97.798,Z 399.928,A -85,B 0,C 180,E1 -29710.872,E2 -29710.872} C_VEL
LIN {X 0,Y 99.069,Z 403.573,A -85,B 0,C 180,E1 -29717.403,E2 -29717.403} C_VEL
LIN {X 0,Y 100.518,Z 407.234,A -85,B 0,C 180,E1 -29721.755,E2 -29721.755} C_VEL
LIN {X 0,Y 102.397,Z 412.309,A -85,B 0,C 180,E1 -29726.041,E2 -29726.041} C_VEL
LIN {X 0,Y 102.71,Z 413.255,A -85,B 0,C 180,E1 -29726.68,E2 -29726.68} C_VEL
LIN {X 0,Y 100.258,Z 434.658,A -85,B 0,C 180,E1 -29727.594,E2 -29727.594} C_VEL
LIN {X 0,Y 97.368,Z 448.405,A -85,B 0,C 180,E1 -29728.583,E2 -29728.583} C_VEL
LIN {X 0,Y 93.915,Z 459.597,A -85,B 0,C 180,E1 -29729.778,E2 -29729.778} C_VEL
LIN {X 0,Y 91.603,Z 465.024,A -85,B 0,C 180,E1 -29730.057,E2 -29730.057} C_VEL
LIN {X 0,Y 86.594,Z 473.575,A -85,B 0,C 180,E1 -29729.621,E2 -29729.621} C_VEL
LIN {X 0,Y 80.967,Z 481.729,A -85,B 0,C 180,E1 -29729.374,E2 -29729.374} C_VEL
LIN {X 0,Y 77.678,Z 486.529,A -85,B 0,C 180,E1 -29730.087,E2 -29730.087} C_VEL
LIN {X 0,Y 71.15,Z 495.766,A -85,B 0,C 180,E1 -29732.906,E2 -29732.906} C_VEL
LIN {X 0,Y 63.718,Z 504.691,A -85,B 0,C 180,E1 -29736.906,E2 -29736.906} C_VEL
LIN {X 0,Y 55.321,Z 513.402,A -85,B 0,C 180,E1 -29743.077,E2 -29743.077} C_VEL
LIN {X 0,Y 47.751,Z 520.346,A -85,B 0,C 180,E1 -29751.284,E2 -29751.284} C_VEL
LIN {X 0,Y 40.404,Z 526.727,A -85,B 0,C 180,E1 -29764.228,E2 -29764.228} C_VEL
LIN {X 0,Y 36.237,Z 530.919,A -85,B 0,C 180,E1 -29778.821,E2 -29778.821} C_VEL
LIN {X 0,Y 34.602,Z 533.165,A -85,B 0,C 180,E1 -29790.004,E2 -29790.004} C_VEL
LIN {X 0,Y 34.082,Z 534.933,A -85,B 0,C 180,E1 -29801.905,E2 -29801.905} C_VEL
LIN {X 0,Y 37.117,Z 537.244,A -85,B 0,C 180,E1 -29824.618,E2 -29824.618} C_VEL
LIN {X 0,Y 42.715,Z 537.901,A -85,B 0,C 180,E1 -29838.845,E2 -29838.845} C_VEL
LIN {X 0,Y 49.37,Z 537.615,A -85,B 0,C 180,E1 -29848.667,E2 -29848.667} C_VEL
LIN {X 0,Y 54.693,Z 536.94,A -85,B 0,C 180,E1 -29854.097,E2 -29854.097} C_VEL
LIN {X 0,Y 64.098,Z 534.939,A -85,B 0,C 180,E1 -29860.797,E2 -29860.797} C_VEL
LIN {X 0,Y 75.878,Z 531.1,A -85,B 0,C 180,E1 -29866.548,E2 -29866.548} C_VEL
LIN {X 0,Y 85.649,Z 526.83,A -85,B 0,C 180,E1 -29869.96,E2 -29869.96} C_VEL
LIN {X 0,Y 95.664,Z 521.328,A -85,B 0,C 180,E1 -29872.659,E2 -29872.659} C_VEL
LIN {X 0,Y 105.853,Z 514.411,A -85,B 0,C 180,E1 -29874.824,E2 -29874.824} C_VEL
LIN {X 0,Y 115.449,Z 506.38,A -85,B 0,C 180,E1 -29876.511,E2 -29876.511} C_VEL
LIN {X 0,Y 124.828,Z 496.697,A -85,B 0,C 180,E1 -29877.951,E2 -29877.951} C_VEL
LIN {X 0,Y 132.673,Z 486.752,A -85,B 0,C 180,E1 -29879.046,E2 -29879.046} C_VEL
LIN {X 0,Y 139.525,Z 476.023,A -85,B 0,C 180,E1 -29879.843,E2 -29879.843} C_VEL
LIN {X 0,Y 145.519,Z 464.002,A -85,B 0,C 180,E1 -29880.557,E2 -29880.557} C_VEL
LIN {X 0,Y 146.195,Z 462.451,A -85,B 0,C 180,E1 -29880.625,E2 -29880.625} C_VEL
LIN {X 0,Y 146.951,Z 460.546,A -85,B 0,C 180,E1 -29880.923,E2 -29880.923} C_VEL
LIN {X 0,Y 147.027,Z 459.837,A -85,B 0,C 180,E1 -29882.74,E2 -29882.74} C_VEL
LIN {X 0,Y 146.985,Z 459.914,A -85,B 0,C 180,E1 -29885.488,E2 -29885.488} C_VEL
LIN {X 0,Y 147.038,Z 460.83,A -85,B 0,C 180,E1 -29888.59,E2 -29888.59} C_VEL
LIN {X 0,Y 146.185,Z 462.998,A -85,B 0,C 180,E1 -29888.793,E2 -29888.793} C_VEL
LIN {X 0,Y 140.629,Z 474.555,A -85,B 0,C 180,E1 -29889.239,E2 -29889.239} C_VEL
LIN {X 0,Y 133.74,Z 485.83,A -85,B 0,C 180,E1 -29889.831,E2 -29889.831} C_VEL
LIN {X 0,Y 126.046,Z 496.002,A -85,B 0,C 180,E1 -29890.661,E2 -29890.661} C_VEL
LIN {X 0,Y 116.662,Z 505.982,A -85,B 0,C 180,E1 -29891.777,E2 -29891.777} C_VEL
LIN {X 0,Y 106.527,Z 514.781,A -85,B 0,C 180,E1 -29893.313,E2 -29893.313} C_VEL
LIN {X 0,Y 96.509,Z 521.853,A -85,B 0,C 180,E1 -29895.222,E2 -29895.222} C_VEL
LIN {X 0,Y 84.995,Z 528.332,A -85,B 0,C 180,E1 -29898.025,E2 -29898.025} C_VEL
LIN {X 0,Y 75.388,Z 532.636,A -85,B 0,C 180,E1 -29901.209,E2 -29901.209} C_VEL
LIN {X 0,Y 67.729,Z 535.413,A -85,B 0,C 180,E1 -29904.525,E2 -29904.525} C_VEL
LIN {X 0,Y 57.331,Z 538.211,A -85,B 0,C 180,E1 -29910.891,E2 -29910.891} C_VEL
LIN {X 0,Y 46.786,Z 539.886,A -85,B 0,C 180,E1 -29921.311,E2 -29921.311} C_VEL
LIN {X 0,Y 42.304,Z 540.156,A -85,B 0,C 180,E1 -29928.35,E2 -29928.35} C_VEL
LIN {X 0,Y 36.061,Z 539.478,A -85,B 0,C 180,E1 -29947.055,E2 -29947.055} C_VEL
LIN {X 0,Y 34.611,Z 538.563,A -85,B 0,C 180,E1 -29958.28,E2 -29958.28} C_VEL
LIN {X 0,Y 34.379,Z 537.252,A -85,B 0,C 180,E1 -29969.996,E2 -29969.996} C_VEL
LIN {X 0,Y 35.13,Z 534.356,A -85,B 0,C 180,E1 -29987.458,E2 -29987.458} C_VEL
LIN {X 0,Y 38.517,Z 530.395,A -85,B 0,C 180,E1 -30003.183,E2 -30003.183} C_VEL
LIN {X 0,Y 45.357,Z 524.287,A -85,B 0,C 180,E1 -30017.387,E2 -30017.387} C_VEL
LIN {X 0,Y 52.801,Z 517.577,A -85,B 0,C 180,E1 -30026.288,E2 -30026.288} C_VEL
LIN {X 0,Y 59.373,Z 511.022,A -85,B 0,C 180,E1 -30031.86,E2 -30031.86} C_VEL
LIN {X 0,Y 67.049,Z 502.463,A -85,B 0,C 180,E1 -30036.509,E2 -30036.509} C_VEL
LIN {X 0,Y 74.769,Z 492.377,A -85,B 0,C 180,E1 -30040.038,E2 -30040.038} C_VEL
LIN {X 0,Y 81.116,Z 482.38,A -85,B 0,C 180,E1 -30042.368,E2 -30042.368} C_VEL
LIN {X 0,Y 86.806,Z 471.523,A -85,B 0,C 180,E1 -30044.026,E2 -30044.026} C_VEL
LIN {X 0,Y 91.308,Z 460.671,A -85,B 0,C 180,E1 -30045.218,E2 -30045.218} C_VEL
LIN {X 0,Y 95.332,Z 447.67,A -85,B 0,C 180,E1 -30046.2,E2 -30046.2} C_VEL
LIN {X 0,Y 97.787,Z 435.605,A -85,B 0,C 180,E1 -30046.849,E2 -30046.849} C_VEL
LIN {X 0,Y 100.017,Z 416.93,A -85,B 0,C 180,E1 -30047.44,E2 -30047.44} C_VEL
LIN {X 0,Y 98.702,Z 412.829,A -85,B 0,C 180,E1 -30051.167,E2 -30051.167} C_VEL
LIN {X 0,Y 97.458,Z 408.934,A -85,B 0,C 180,E1 -30056.123,E2 -30056.123} C_VEL
LIN {X 0,Y 96.816,Z 406.306,A -85,B 0,C 180,E1 -30061.039,E2 -30061.039} C_VEL
LIN {X 0,Y 96.77,Z 406.554,A -85,B 0,C 180,E1 -30069.404,E2 -30069.404} C_VEL
LIN {X 0,Y 97.798,Z 410.267,A -85,B 0,C 180,E1 -30076.168,E2 -30076.168} C_VEL
LIN {X 0,Y 98.918,Z 413.576,A -85,B 0,C 180,E1 -30080.129,E2 -30080.129} C_VEL
LIN {X 0,Y 99.965,Z 416.842,A -85,B 0,C 180,E1 -30083.041,E2 -30083.041} C_VEL
LIN {X 0,Y 97.542,Z 436.228,A -85,B 0,C 180,E1 -30083.821,E2 -30083.821} C_VEL
LIN {X 0,Y 94.906,Z 448.164,A -85,B 0,C 180,E1 -30084.616,E2 -30084.616} C_VEL
LIN {X 0,Y 91.18,Z 459.897,A -85,B 0,C 180,E1 -30085.734,E2 -30085.734} C_VEL
LIN {X 0,Y 85.991,Z 471.944,A -85,B 0,C 180,E1 -30087.281,E2 -30087.281} C_VEL
LIN {X 0,Y 79.605,Z 483.447,A -85,B 0,C 180,E1 -30089.334,E2 -30089.334} C_VEL
LIN {X 0,Y 77.678,Z 486.529,A -85,B 0,C 180,E1 -30090.087,E2 -30090.087} C_VEL
LIN {X 0,Y 74.22,Z 491.259,A -85,B 0,C 180,E1 -30090.953,E2 -30090.953} C_VEL
LIN {X 0,Y 67.48,Z 498.546,A -85,B 0,C 180,E1 -30091.311,E2 -30091.311} C_VEL
LIN {X 0,Y 60.272,Z 505.287,A -85,B 0,C 180,E1 -30091.939,E2 -30091.939} C_VEL
LIN {X 0,Y 56.135,Z 509.132,A -85,B 0,C 180,E1 -30093.503,E2 -30093.503} C_VEL
LIN {X 0,Y 47.923,Z 516.575,A -85,B 0,C 180,E1 -30099.659,E2 -30099.659} C_VEL
LIN {X 0,Y 41.177,Z 521.979,A -85,B 0,C 180,E1 -30106.949,E2 -30106.949} C_VEL
LIN {X 0,Y 34.157,Z 527.281,A -85,B 0,C 180,E1 -30119.049,E2 -30119.049} C_VEL
LIN {X 0,Y 29.278,Z 531.41,A -85,B 0,C 180,E1 -30136.116,E2 -30136.116} C_VEL
LIN {X 0,Y 27.398,Z 533.605,A -85,B 0,C 180,E1 -30150.005,E2 -30150.005} C_VEL
LIN {X 0,Y 27.058,Z 535.335,A -85,B 0,C 180,E1 -30165.06,E2 -30165.06} C_VEL
LIN {X 0,Y 31.428,Z 537.586,A -85,B 0,C 180,E1 -30192.14,E2 -30192.14} C_VEL
LIN {X 0,Y 37.523,Z 538.155,A -85,B 0,C 180,E1 -30205.816,E2 -30205.816} C_VEL
LIN {X 0,Y 45.994,Z 537.842,A -85,B 0,C 180,E1 -30216.472,E2 -30216.472} C_VEL
LIN {X 0,Y 51.927,Z 537.131,A -85,B 0,C 180,E1 -30221.342,E2 -30221.342} C_VEL
LIN {X 0,Y 61.159,Z 535.285,A -85,B 0,C 180,E1 -30226.714,E2 -30226.714} C_VEL
LIN {X 0,Y 71.179,Z 532.357,A -85,B 0,C 180,E1 -30230.892,E2 -30230.892} C_VEL
LIN {X 0,Y 81.276,Z 528.403,A -85,B 0,C 180,E1 -30233.954,E2 -30233.954} C_VEL
LIN {X 0,Y 91.554,Z 523.257,A -85,B 0,C 180,E1 -30236.328,E2 -30236.328} C_VEL
LIN {X 0,Y 101.957,Z 516.719,A -85,B 0,C 180,E1 -30238.208,E2 -30238.208} C_VEL
LIN {X 0,Y 112.451,Z 508.537,A -85,B 0,C 180,E1 -30239.727,E2 -30239.727} C_VEL
LIN {X 0,Y 121.248,Z 500.133,A -85,B 0,C 180,E1 -30240.867,E2 -30240.867} C_VEL
LIN {X 0,Y 129.205,Z 490.913,A -85,B 0,C 180,E1 -30241.8,E2 -30241.8} C_VEL
LIN {X 0,Y 136.663,Z 480.235,A -85,B 0,C 180,E1 -30242.533,E2 -30242.533} C_VEL
LIN {X 0,Y 143.347,Z 468.133,A -85,B 0,C 180,E1 -30243.188,E2 -30243.188} C_VEL
LIN {X 0,Y 144.189,Z 466.381,A -85,B 0,C 180,E1 -30243.423,E2 -30243.423} C_VEL
LIN {X 0,Y 144.18,Z 466.498,A -85,B 0,C 180,E1 -30245.595,E2 -30245.595} C_VEL
LIN {X 0,Y 143.634,Z 467.744,A -85,B 0,C 180,E1 -30246.135,E2 -30246.135} C_VEL
LIN {X 0,Y 137.062,Z 479.817,A -85,B 0,C 180,E1 -30246.545,E2 -30246.545} C_VEL
LIN {X 0,Y 129.245,Z 491.155,A -85,B 0,C 180,E1 -30247.07,E2 -30247.07} C_VEL
LIN {X 0,Y 120.6,Z 501.167,A -85,B 0,C 180,E1 -30247.823,E2 -30247.823} C_VEL
LIN {X 0,Y 111.981,Z 509.384,A -85,B 0,C 180,E1 -30248.7,E2 -30248.7} C_VEL
LIN {X 0,Y 101.71,Z 517.45,A -85,B 0,C 180,E1 -30250.045,E2 -30250.045} C_VEL
LIN {X 0,Y 93.189,Z 522.949,A -85,B 0,C 180,E1 -30251.354,E2 -30251.354} C_VEL
LIN {X 0,Y 83.07,Z 528.347,A -85,B 0,C 180,E1 -30253.354,E2 -30253.354} C_VEL
LIN {X 0,Y 73.115,Z 532.587,A -85,B 0,C 180,E1 -30256.002,E2 -30256.002} C_VEL
LIN {X 0,Y 64.263,Z 535.54,A -85,B 0,C 180,E1 -30259.154,E2 -30259.154} C_VEL
LIN {X 0,Y 54.024,Z 538.043,A -85,B 0,C 180,E1 -30264.401,E2 -30264.401} C_VEL
LIN {X 0,Y 42.416,Z 539.662,A -85,B 0,C 180,E1 -30274.054,E2 -30274.054} C_VEL
LIN {X 0,Y 37.277,Z 539.886,A -85,B 0,C 180,E1 -30281.044,E2 -30281.044} C_VEL
LIN {X 0,Y 29.634,Z 539.143,A -85,B 0,C 180,E1 -30301.68,E2 -30301.68} C_VEL
LIN {X 0,Y 27.68,Z 538.2,A -85,B 0,C 180,E1 -30315.286,E2 -30315.286} C_VEL
LIN {X 0,Y 27.272,Z 536.852,A -85,B 0,C 180,E1 -30329.995,E2 -30329.995} C_VEL
LIN {X 0,Y 28.414,Z 533.903,A -85,B 0,C 180,E1 -30351.773,E2 -30351.773} C_VEL
LIN {X 0,Y 32.77,Z 529.877,A -85,B 0,C 180,E1 -30370.039,E2 -30370.039} C_VEL
LIN {X 0,Y 40.852,Z 523.668,A -85,B 0,C 180,E1 -30384.795,E2 -30384.795} C_VEL
LIN {X 0,Y 49.179,Z 516.885,A -85,B 0,C 180,E1 -30393.243,E2 -30393.243} C_VEL
LIN {X 0,Y 54.813,Z 511.742,A -85,B 0,C 180,E1 -30397.376,E2 -30397.376} C_VEL
LIN {X 0,Y 62.931,Z 503.374,A -85,B 0,C 180,E1 -30401.662,E2 -30401.662} C_VEL
LIN {X 0,Y 70.992,Z 493.523,A -85,B 0,C 180,E1 -30404.835,E2 -30404.835} C_VEL
LIN {X 0,Y 77.593,Z 483.88,A -85,B 0,C 180,E1 -30406.817,E2 -30406.817} C_VEL
LIN {X 0,Y 83.434,Z 473.505,A -85,B 0,C 180,E1 -30408.291,E2 -30408.291} C_VEL
LIN {X 0,Y 88.487,Z 462.272,A -85,B 0,C 180,E1 -30409.342,E2 -30409.342} C_VEL
LIN {X 0,Y 92.89,Z 448.902,A -85,B 0,C 180,E1 -30410.234,E2 -30410.234} C_VEL
LIN {X 0,Y 95.615,Z 436.503,A -85,B 0,C 180,E1 -30410.841,E2 -30410.841} C_VEL
LIN {X 0,Y 97.639,Z 420.604,A -85,B 0,C 180,E1 -30411.341,E2 -30411.341} C_VEL
LIN {X 0,Y 96.662,Z 417.129,A -85,B 0,C 180,E1 -30415.307,E2 -30415.307} C_VEL
LIN {X 0,Y 96.117,Z 414.922,A -85,B 0,C 180,E1 -30418.69,E2 -30418.69} C_VEL
LIN {X 0,Y 95.888,Z 413.312,A -85,B 0,C 180,E1 -30421.574,E2 -30421.574} C_VEL
LIN {X 0,Y 95.828,Z 413.557,A -85,B 0,C 180,E1 -30428.699,E2 -30428.699} C_VEL
LIN {X 0,Y 96.548,Z 416.848,A -85,B 0,C 180,E1 -30434.759,E2 -30434.759} C_VEL
LIN {X 0,Y 97.513,Z 420.236,A -85,B 0,C 180,E1 -30438.834,E2 -30438.834} C_VEL
LIN {X 0,Y 97.607,Z 420.601,A -85,B 0,C 180,E1 -30439.174,E2 -30439.174} C_VEL
LIN {X 0,Y 95.313,Z 437.572,A -85,B 0,C 180,E1 -30439.842,E2 -30439.842} C_VEL
LIN {X 0,Y 92.207,Z 450.527,A -85,B 0,C 180,E1 -30440.654,E2 -30440.654} C_VEL
LIN {X 0,Y 87.928,Z 462.656,A -85,B 0,C 180,E1 -30441.7,E2 -30441.7} C_VEL
LIN {X 0,Y 82.961,Z 473.359,A -85,B 0,C 180,E1 -30442.893,E2 -30442.893} C_VEL
LIN {X 0,Y 76.394,Z 484.638,A -85,B 0,C 180,E1 -30444.711,E2 -30444.711} C_VEL
LIN {X 0,Y 69.17,Z 494.777,A -85,B 0,C 180,E1 -30447.252,E2 -30447.252} C_VEL
LIN {X 0,Y 61.28,Z 503.914,A -85,B 0,C 180,E1 -30450.672,E2 -30450.672} C_VEL
LIN {X 0,Y 56.135,Z 509.132,A -85,B 0,C 180,E1 -30453.503,E2 -30453.503} C_VEL
LIN {X 0,Y 51.886,Z 512.823,A -85,B 0,C 180,E1 -30455.435,E2 -30455.435} C_VEL
LIN {X 0,Y 43.861,Z 518.346,A -85,B 0,C 180,E1 -30457.708,E2 -30457.708} C_VEL
LIN {X 0,Y 35.583,Z 523.317,A -85,B 0,C 180,E1 -30461.31,E2 -30461.31} C_VEL
LIN {X 0,Y 31.139,Z 525.979,A -85,B 0,C 180,E1 -30466.161,E2 -30466.161} C_VEL
LIN {X 0,Y 24.104,Z 530.645,A -85,B 0,C 180,E1 -30484.072,E2 -30484.072} C_VEL
LIN {X 0,Y 21.651,Z 532.564,A -85,B 0,C 180,E1 -30496.846,E2 -30496.846} C_VEL
LIN {X 0,Y 20.161,Z 535.737,A -85,B 0,C 180,E1 -30530.409,E2 -30530.409} C_VEL
LIN {X 0,Y 22.443,Z 537.034,A -85,B 0,C 180,E1 -30548.786,E2 -30548.786} C_VEL
LIN {X 0,Y 26.51,Z 537.915,A -85,B 0,C 180,E1 -30562.693,E2 -30562.693} C_VEL
LIN {X 0,Y 33.134,Z 538.411,A -85,B 0,C 180,E1 -30574.902,E2 -30574.902} C_VEL
LIN {X 0,Y 43.6,Z 538.069,A -85,B 0,C 180,E1 -30585.284,E2 -30585.284} C_VEL
LIN {X 0,Y 50.072,Z 537.306,A -85,B 0,C 180,E1 -30589.281,E2 -30589.281} C_VEL
LIN {X 0,Y 58.863,Z 535.643,A -85,B 0,C 180,E1 -30593.144,E2 -30593.144} C_VEL
LIN {X 0,Y 70.394,Z 532.423,A -85,B 0,C 180,E1 -30596.767,E2 -30596.767} C_VEL
LIN {X 0,Y 80.834,Z 528.398,A -85,B 0,C 180,E1 -30599.089,E2 -30599.089} C_VEL
LIN {X 0,Y 93.141,Z 522.143,A -85,B 0,C 180,E1 -30601.146,E2 -30601.146} C_VEL
LIN {X 0,Y 103.763,Z 515.289,A -85,B 0,C 180,E1 -30602.493,E2 -30602.493} C_VEL
LIN {X 0,Y 114.255,Z 506.853,A -85,B 0,C 180,E1 -30603.601,E2 -30603.601} C_VEL
